(* CODESYS project BaseCodesys

Project tree, tasks and I/O mapping:
  Device : Berghof MC-PI SoftMotion Control , Berghof Automation GmbH, version 1.2.1.0
    application Application
      libraries: Standard, 3.5.18.0 (System); VisuDialogs, * (System)
      task EtherCAT_Task (cyclic, interval 1 ms, priority 0) calls PLC_PRG, POU
      task VISU_TASK (cyclic, interval 100 ms, priority 31) calls VisuElems.Visu_Prg
      program PLC_PRG [LD]
      trace Suivi (task EtherCAT_Task): PLC_PRG.MC_ReadActualPosition_0.Position
      Symbols
    EtherCAT_Master_SoftMotion : EtherCAT Master SoftMotion, 3S - Smart Software Solutions GmbH, version 4.4.0.0
        settings: MasterCycleTime = 1000; SlaveAutoRestart = True; NetworkName = 'eth0'; NetworkName = "eth0"; SrcAddress1 = 58463; SrcAddress2 = 30116746
      SC6_1 : SI6_SC6_DoubleAx_SoftMotion, STOEBER ANTRIEBSTECHNIK GmbH & Co. KG, version 4.5.0.0
          settings: ModularDevice = True; Number of Outputs = 0; Number of Inputs = 0; Number of Infos about Outputs = 0; Number of Infos about Inputs = 0; EnableExpertSettings = True; MDP_InputOffsets = [0,0,232]; MDP_OutputOffsets = [0,0,184]; StationAlias = 1002; Optional = False; DeviceIdenticationADO = 0; DeviceIdenticationMode = 0; Sync.Length = 46; Sync.Length = 58; FMMU.Length = 46; FMMU.Length = 58; Number of RxPDOs of the Slave = 2; Number of TxPDOs of the Slave = 2; DC sync0 cycletime = 1000; DC sync1 cycletime = 1000; EoEEnabled = True; EoEVirtualMACID = [16#02,16#01,16#05,16#10,16#03,16#E9]; EoEIPPortEnabled = False; EoEIPAddress = [16#00,16#00,16#00,16#00]; EoESubnetMask = [16#00,16#00,16#00,16#00]; EoEDefaultGateway = [16#00,16#00,16#00,16#00]; EoEDNSServer = [16#00,16#00,16#00,16#00]; EoEDNSName = 'SC6_1'; RxTxPdo.NumberofExcludes = 0; RxTxPdo.NumberofEntries = 8; RxTxPdo.Index = 16#1600; RxTxPdo.Fixed = False; RxTxPdo.Mandatory = False; RxTxPdo.Virtual = False; RxTxPdo.Sm = 2; RxTxPdo.Su = 0; RxTxPdo.Name = 'Axis A to Slave'; RxTxPdo.DependOnSlot = False; RxTxPdo.DependOnSlotGroup = False; RxTxPdo.OverwrittenByModule = True;
            A515 Controlword.Index = 16#6040; A515 Controlword.SubIndex = 0; A515 Controlword.Size = 16; A515 Controlword.Offset = 0; A515 Controlword.DependOnSlot = False; A515 Controlword.DependOnSlotGroup = False; A541 Modes of operation.Index = 16#6060; A541 Modes of operation.SubIndex = 0; A541 Modes of operation.Size = 8; A541 Modes of operation.Offset = 0; A541 Modes of operation.DependOnSlot = False; A541 Modes of operation.DependOnSlotGroup = False; A567 Target position.Index = 16#607A; A567 Target position.SubIndex = 0; A567 Target position.Size = 32; A567 Target position.Offset = 0; A567 Target position.DependOnSlot = False; A567 Target position.DependOnSlotGroup = False; A638 Target velocity.Index = 16#60FF; A638 Target velocity.SubIndex = 0; A638 Target velocity.Size = 32; A638 Target velocity.Offset = 0; A638 Target velocity.DependOnSlot = False; A638 Target velocity.DependOnSlotGroup = False; A592 Velocity offset.Index = 16#60B1; A592 Velocity offset.SubIndex = 0; A592 Velocity offset.Size = 32; A592 Velocity offset.Offset = 0; A592 Velocity offset.DependOnSlot = False; A592 Velocity offset.DependOnSlotGroup = False; A593 Torque offset.Index = 16#60B2; A593 Torque offset.SubIndex = 0; A593 Torque offset.Size = 16; A593 Torque offset.Offset = 0; A593 Torque offset.DependOnSlot = False; A593 Torque offset.DependOnSlotGroup = False; A558 Target torque.Index = 16#6071; A558 Target torque.SubIndex = 0; A558 Target torque.Size = 16; A558 Target torque.Offset = 0;
            A558 Target torque.DependOnSlot = False; A558 Target torque.DependOnSlotGroup = False; A637 Digital outputs.Index = 16#60FE; A637 Digital outputs.SubIndex = 1; A637 Digital outputs.Size = 32; A637 Digital outputs.Offset = 0; A637 Digital outputs.DependOnSlot = False; A637 Digital outputs.DependOnSlotGroup = False; RxTxPdo.NumberofExcludes = 0; RxTxPdo.NumberofEntries = 8; RxTxPdo.Index = 16#1601; RxTxPdo.Fixed = False; RxTxPdo.Mandatory = False; RxTxPdo.Virtual = False; RxTxPdo.Sm = 2; RxTxPdo.Su = 0; RxTxPdo.Name = 'Axis B to Slave'; RxTxPdo.DependOnSlot = False; RxTxPdo.DependOnSlotGroup = False; RxTxPdo.OverwrittenByModule = True; 2.A515 Controlword.Index = 16#6840; 2.A515 Controlword.SubIndex = 0; 2.A515 Controlword.Size = 16; 2.A515 Controlword.Offset = 0; 2.A515 Controlword.DependOnSlot = False; 2.A515 Controlword.DependOnSlotGroup = False; 2.A541 Modes of operation.Index = 16#6860; 2.A541 Modes of operation.SubIndex = 0; 2.A541 Modes of operation.Size = 8; 2.A541 Modes of operation.Offset = 0; 2.A541 Modes of operation.DependOnSlot = False; 2.A541 Modes of operation.DependOnSlotGroup = False; 2.A567 Target position.Index = 16#687A; 2.A567 Target position.SubIndex = 0; 2.A567 Target position.Size = 32; 2.A567 Target position.Offset = 0; 2.A567 Target position.DependOnSlot = False; 2.A567 Target position.DependOnSlotGroup = False; 2.A638 Target velocity.Index = 16#68FF; 2.A638 Target velocity.SubIndex = 0;
            2.A638 Target velocity.Size = 32; 2.A638 Target velocity.Offset = 0; 2.A638 Target velocity.DependOnSlot = False; 2.A638 Target velocity.DependOnSlotGroup = False; 2.A592 Velocity offset.Index = 16#68B1; 2.A592 Velocity offset.SubIndex = 0; 2.A592 Velocity offset.Size = 32; 2.A592 Velocity offset.Offset = 0; 2.A592 Velocity offset.DependOnSlot = False; 2.A592 Velocity offset.DependOnSlotGroup = False; 2.A593 Torque offset.Index = 16#68B2; 2.A593 Torque offset.SubIndex = 0; 2.A593 Torque offset.Size = 16; 2.A593 Torque offset.Offset = 0; 2.A593 Torque offset.DependOnSlot = False; 2.A593 Torque offset.DependOnSlotGroup = False; 2.A558 Target torque.Index = 16#6871; 2.A558 Target torque.SubIndex = 0; 2.A558 Target torque.Size = 16; 2.A558 Target torque.Offset = 0; 2.A558 Target torque.DependOnSlot = False; 2.A558 Target torque.DependOnSlotGroup = False; 2.A637 Digital outputs.Index = 16#68FE; 2.A637 Digital outputs.SubIndex = 1; 2.A637 Digital outputs.Size = 32; 2.A637 Digital outputs.Offset = 0; 2.A637 Digital outputs.DependOnSlot = False; 2.A637 Digital outputs.DependOnSlotGroup = False; RxTxPdo.NumberofExcludes = 0; RxTxPdo.NumberofEntries = 10; RxTxPdo.Index = 16#1A00; RxTxPdo.Fixed = False; RxTxPdo.Mandatory = False; RxTxPdo.Virtual = False; RxTxPdo.Sm = 3; RxTxPdo.Su = 0; RxTxPdo.Name = 'Axis A to Master'; RxTxPdo.DependOnSlot = False; RxTxPdo.DependOnSlotGroup = False; RxTxPdo.OverwrittenByModule = True;
            A516 Statusword.Index = 16#6041; A516 Statusword.SubIndex = 0; A516 Statusword.Size = 16; A516 Statusword.Offset = 0; A516 Statusword.DependOnSlot = False; A516 Statusword.DependOnSlotGroup = False; A542 Modes of operation display.Index = 16#6061; A542 Modes of operation display.SubIndex = 0; A542 Modes of operation display.Size = 8; A542 Modes of operation display.Offset = 0; A542 Modes of operation display.DependOnSlot = False; A542 Modes of operation display.DependOnSlotGroup = False; A545 Position actual value.Index = 16#6064; A545 Position actual value.SubIndex = 0; A545 Position actual value.Size = 32; A545 Position actual value.Offset = 0; A545 Position actual value.DependOnSlot = False; A545 Position actual value.DependOnSlotGroup = False; A553 Velocity actual value.Index = 16#606C; A553 Velocity actual value.SubIndex = 0; A553 Velocity actual value.Size = 32; A553 Velocity actual value.Offset = 0; A553 Velocity actual value.DependOnSlot = False; A553 Velocity actual value.DependOnSlotGroup = False; A564 Torque actual value.Index = 16#6077; A564 Torque actual value.SubIndex = 0; A564 Torque actual value.Size = 16; A564 Torque actual value.Offset = 0; A564 Torque actual value.DependOnSlot = False; A564 Torque actual value.DependOnSlotGroup = False; A632 Following error actual value.Index = 16#60F4; A632 Following error actual value.SubIndex = 0; A632 Following error actual value.Size = 32; A632 Following error actual value.Offset = 0; A632 Following error actual value.DependOnSlot = False; A632 Following error actual value.DependOnSlotGroup = False; A636 Digital inputs.Index = 16#60FD; A636 Digital inputs.SubIndex = 0; A636 Digital inputs.Size = 32; A636 Digital inputs.Offset = 0;
            A636 Digital inputs.DependOnSlot = False; A636 Digital inputs.DependOnSlotGroup = False; A620 Additional position actual value / 1st value.Index = 16#60E4; A620 Additional position actual value / 1st value.SubIndex = 1; A620 Additional position actual value / 1st value.Size = 32; A620 Additional position actual value / 1st value.Offset = 0; A620 Additional position actual value / 1st value.DependOnSlot = False; A620 Additional position actual value / 1st value.DependOnSlotGroup = False; E201 Statuswort 2.Index = 16#28C9; E201 Statuswort 2.SubIndex = 0; E201 Statuswort 2.Size = 16; E201 Statuswort 2.Offset = 0; E201 Statuswort 2.DependOnSlot = False; E201 Statuswort 2.DependOnSlotGroup = False; A67 User Statuswort.Index = 16#2043; A67 User Statuswort.SubIndex = 0; A67 User Statuswort.Size = 16; A67 User Statuswort.Offset = 0; A67 User Statuswort.DependOnSlot = False; A67 User Statuswort.DependOnSlotGroup = False; RxTxPdo.NumberofExcludes = 0; RxTxPdo.NumberofEntries = 10; RxTxPdo.Index = 16#1A01; RxTxPdo.Fixed = False; RxTxPdo.Mandatory = False; RxTxPdo.Virtual = False; RxTxPdo.Sm = 3; RxTxPdo.Su = 0; RxTxPdo.Name = 'Axis B to Master'; RxTxPdo.DependOnSlot = False; RxTxPdo.DependOnSlotGroup = False; RxTxPdo.OverwrittenByModule = True; 2.A516 Statusword.Index = 16#6841; 2.A516 Statusword.SubIndex = 0; 2.A516 Statusword.Size = 16; 2.A516 Statusword.Offset = 0; 2.A516 Statusword.DependOnSlot = False; 2.A516 Statusword.DependOnSlotGroup = False; 2.A542 Modes of operation display.Index = 16#6861; 2.A542 Modes of operation display.SubIndex = 0;
            2.A542 Modes of operation display.Size = 8; 2.A542 Modes of operation display.Offset = 0; 2.A542 Modes of operation display.DependOnSlot = False; 2.A542 Modes of operation display.DependOnSlotGroup = False; 2.A545 Position actual value.Index = 16#6864; 2.A545 Position actual value.SubIndex = 0; 2.A545 Position actual value.Size = 32; 2.A545 Position actual value.Offset = 0; 2.A545 Position actual value.DependOnSlot = False; 2.A545 Position actual value.DependOnSlotGroup = False; 2.A553 Velocity actual value.Index = 16#686C; 2.A553 Velocity actual value.SubIndex = 0; 2.A553 Velocity actual value.Size = 32; 2.A553 Velocity actual value.Offset = 0; 2.A553 Velocity actual value.DependOnSlot = False; 2.A553 Velocity actual value.DependOnSlotGroup = False; 2.A564 Torque actual value.Index = 16#6877; 2.A564 Torque actual value.SubIndex = 0; 2.A564 Torque actual value.Size = 16; 2.A564 Torque actual value.Offset = 0; 2.A564 Torque actual value.DependOnSlot = False; 2.A564 Torque actual value.DependOnSlotGroup = False; 2.A632 Following error actual value.Index = 16#68F4; 2.A632 Following error actual value.SubIndex = 0; 2.A632 Following error actual value.Size = 32; 2.A632 Following error actual value.Offset = 0; 2.A632 Following error actual value.DependOnSlot = False; 2.A632 Following error actual value.DependOnSlotGroup = False; 2.636 Digital inputs.Index = 16#68FD; 2.636 Digital inputs.SubIndex = 0; 2.636 Digital inputs.Size = 32; 2.636 Digital inputs.Offset = 0; 2.636 Digital inputs.DependOnSlot = False; 2.636 Digital inputs.DependOnSlotGroup = False; 2.A620 Additional position actual value / 1st value.Index = 16#68E4; 2.A620 Additional position actual value / 1st value.SubIndex = 1; 2.A620 Additional position actual value / 1st value.Size = 32; 2.A620 Additional position actual value / 1st value.Offset = 0; 2.A620 Additional position actual value / 1st value.DependOnSlot = False; 2.A620 Additional position actual value / 1st value.DependOnSlotGroup = False;
            2.E201 Statuswort 2.Index = 16#A8C9; 2.E201 Statuswort 2.SubIndex = 0; 2.E201 Statuswort 2.Size = 16; 2.E201 Statuswort 2.Offset = 0; 2.E201 Statuswort 2.DependOnSlot = False; 2.E201 Statuswort 2.DependOnSlotGroup = False; 2.A67 User Statuswort.Index = 16#A043; 2.A67 User Statuswort.SubIndex = 0; 2.A67 User Statuswort.Size = 16; 2.A67 User Statuswort.Offset = 0; 2.A67 User Statuswort.DependOnSlot = False; 2.A67 User Statuswort.DependOnSlotGroup = False; A515 Controlword.Name = 'A515 Controlword'; A515 Controlword.DataType = 'WORD'; A515 Controlword.Default = ''; A515 Controlword.Comment = ''; A541 Modes of operation.Name = 'A541 Modes of operation'; A541 Modes of operation.DataType = 'SINT'; A541 Modes of operation.Default = ''; A541 Modes of operation.Comment = ''; A567 Target position.Name = 'A567 Target position'; A567 Target position.DataType = 'DINT'; A567 Target position.Default = ''; A567 Target position.Comment = ''; A638 Target velocity.Name = 'A638 Target velocity'; A638 Target velocity.DataType = 'DINT'; A638 Target velocity.Default = ''; A638 Target velocity.Comment = ''; A592 Velocity offset.Name = 'A592 Velocity offset'; A592 Velocity offset.DataType = 'DINT'; A592 Velocity offset.Default = ''; A592 Velocity offset.Comment = ''; A593 Torque offset.Name = 'A593 Torque offset'; A593 Torque offset.DataType = 'INT'; A593 Torque offset.Default = ''; A593 Torque offset.Comment = ''; A558 Target torque.Name = 'A558 Target torque'; A558 Target torque.DataType = 'INT'; A558 Target torque.Default = ''; A558 Target torque.Comment = '';
            A637 Digital outputs.Name = 'A637 Digital outputs'; A637 Digital outputs.DataType = 'DWORD'; A637 Digital outputs.Default = ''; A637 Digital outputs.Comment = ''; 2.A515 Controlword.Name = '2.A515 Controlword'; 2.A515 Controlword.DataType = 'WORD'; 2.A515 Controlword.Default = ''; 2.A515 Controlword.Comment = ''; 2.A541 Modes of operation.Name = '2.A541 Modes of operation'; 2.A541 Modes of operation.DataType = 'SINT'; 2.A541 Modes of operation.Default = ''; 2.A541 Modes of operation.Comment = ''; 2.A567 Target position.Name = '2.A567 Target position'; 2.A567 Target position.DataType = 'DINT'; 2.A567 Target position.Default = ''; 2.A567 Target position.Comment = ''; 2.A638 Target velocity.Name = '2.A638 Target velocity'; 2.A638 Target velocity.DataType = 'DINT'; 2.A638 Target velocity.Default = ''; 2.A638 Target velocity.Comment = ''; 2.A592 Velocity offset.Name = '2.A592 Velocity offset'; 2.A592 Velocity offset.DataType = 'DINT'; 2.A592 Velocity offset.Default = ''; 2.A592 Velocity offset.Comment = ''; 2.A593 Torque offset.Name = '2.A593 Torque offset'; 2.A593 Torque offset.DataType = 'INT'; 2.A593 Torque offset.Default = ''; 2.A593 Torque offset.Comment = ''; 2.A558 Target torque.Name = '2.A558 Target torque'; 2.A558 Target torque.DataType = 'INT'; 2.A558 Target torque.Default = ''; 2.A558 Target torque.Comment = ''; 2.A637 Digital outputs.Name = '2.A637 Digital outputs'; 2.A637 Digital outputs.DataType = 'DWORD'; 2.A637 Digital outputs.Default = ''; 2.A637 Digital outputs.Comment = ''; A516 Statusword.Name = 'A516 Statusword'; A516 Statusword.DataType = 'WORD'; A516 Statusword.Default = ''; A516 Statusword.Comment = '';
            A542 Modes of operation display.Name = 'A542 Modes of operation display'; A542 Modes of operation display.DataType = 'SINT'; A542 Modes of operation display.Default = ''; A542 Modes of operation display.Comment = ''; A545 Position actual value.Name = 'A545 Position actual value'; A545 Position actual value.DataType = 'DINT'; A545 Position actual value.Default = ''; A545 Position actual value.Comment = ''; A553 Velocity actual value.Name = 'A553 Velocity actual value'; A553 Velocity actual value.DataType = 'DINT'; A553 Velocity actual value.Default = ''; A553 Velocity actual value.Comment = ''; A564 Torque actual value.Name = 'A564 Torque actual value'; A564 Torque actual value.DataType = 'INT'; A564 Torque actual value.Default = ''; A564 Torque actual value.Comment = ''; A632 Following error actual value.Name = 'A632 Following error actual value'; A632 Following error actual value.DataType = 'DINT'; A632 Following error actual value.Default = ''; A632 Following error actual value.Comment = ''; A636 Digital inputs.Name = 'A636 Digital inputs'; A636 Digital inputs.DataType = 'DWORD'; A636 Digital inputs.Default = ''; A636 Digital inputs.Comment = ''; A620 Additional position actual value / 1st value.Name = 'A620 Additional position actual value / 1st value'; A620 Additional position actual value / 1st value.DataType = 'DINT'; A620 Additional position actual value / 1st value.Default = ''; A620 Additional position actual value / 1st value.Comment = ''; E201 Statuswort 2.Name = 'E201 Statuswort 2'; E201 Statuswort 2.DataType = 'WORD'; E201 Statuswort 2.Default = ''; E201 Statuswort 2.Comment = ''; A67 User Statuswort.Name = 'A67 User Statuswort'; A67 User Statuswort.DataType = 'WORD'; A67 User Statuswort.Default = ''; A67 User Statuswort.Comment = ''; 2.A516 Statusword.Name = '2.A516 Statusword'; 2.A516 Statusword.DataType = 'WORD'; 2.A516 Statusword.Default = ''; 2.A516 Statusword.Comment = '';
            2.A542 Modes of operation display.Name = '2.A542 Modes of operation display'; 2.A542 Modes of operation display.DataType = 'SINT'; 2.A542 Modes of operation display.Default = ''; 2.A542 Modes of operation display.Comment = ''; 2.A545 Position actual value.Name = '2.A545 Position actual value'; 2.A545 Position actual value.DataType = 'DINT'; 2.A545 Position actual value.Default = ''; 2.A545 Position actual value.Comment = ''; 2.A553 Velocity actual value.Name = '2.A553 Velocity actual value'; 2.A553 Velocity actual value.DataType = 'DINT'; 2.A553 Velocity actual value.Default = ''; 2.A553 Velocity actual value.Comment = ''; 2.A564 Torque actual value.Name = '2.A564 Torque actual value'; 2.A564 Torque actual value.DataType = 'INT'; 2.A564 Torque actual value.Default = ''; 2.A564 Torque actual value.Comment = ''; 2.A632 Following error actual value.Name = '2.A632 Following error actual value'; 2.A632 Following error actual value.DataType = 'DINT'; 2.A632 Following error actual value.Default = ''; 2.A632 Following error actual value.Comment = ''; 2.636 Digital inputs.Name = '2.636 Digital inputs'; 2.636 Digital inputs.DataType = 'DWORD'; 2.636 Digital inputs.Default = ''; 2.636 Digital inputs.Comment = ''; 2.A620 Additional position actual value / 1st value.Name = '2.A620 Additional position actual value / 1st value'; 2.A620 Additional position actual value / 1st value.DataType = 'DINT'; 2.A620 Additional position actual value / 1st value.Default = ''; 2.A620 Additional position actual value / 1st value.Comment = ''; 2.E201 Statuswort 2.Name = '2.E201 Statuswort 2'; 2.E201 Statuswort 2.DataType = 'WORD'; 2.E201 Statuswort 2.Default = ''; 2.E201 Statuswort 2.Comment = ''; 2.A67 User Statuswort.Name = '2.A67 User Statuswort'; 2.A67 User Statuswort.DataType = 'WORD'; 2.A67 User Statuswort.Default = ''; 2.A67 User Statuswort.Comment = ''
        CiA_ControllerBased : xA CBM_SoftMotion, STOEBER ANTRIEBSTECHNIK GmbH & Co. KG, version 4.4.0.0
            settings: Number of Outputs = 8; Number of Inputs = 10; Number of Infos about Outputs = 8; Number of Infos about Inputs = 10; RxTxPdo.Mandatory = False; RxTxPdo.Virtual = False; RxTxPdo.DependOnSlot = False; RxTxPdo.DependOnSlotGroup = False; A515 Controlword.Offset = 0; A515 Controlword.DependOnSlot = False; A515 Controlword.DependOnSlotGroup = False; A541 Modes of operation.Offset = 0; A541 Modes of operation.DependOnSlot = False; A541 Modes of operation.DependOnSlotGroup = False; A567 Target position.Offset = 0; A567 Target position.DependOnSlot = False; A567 Target position.DependOnSlotGroup = False; A638 Target velocity.Offset = 0; A638 Target velocity.DependOnSlot = False; A638 Target velocity.DependOnSlotGroup = False; A592 Velocity offset.Offset = 0; A592 Velocity offset.DependOnSlot = False; A592 Velocity offset.DependOnSlotGroup = False; A593 Torque offset.Offset = 0; A593 Torque offset.DependOnSlot = False; A593 Torque offset.DependOnSlotGroup = False; A558 Target torque.Offset = 0; A558 Target torque.DependOnSlot = False; A558 Target torque.DependOnSlotGroup = False; A637 Digital outputs.Offset = 0; A637 Digital outputs.DependOnSlot = False; A637 Digital outputs.DependOnSlotGroup = False; RxTxPdo.Mandatory = False; RxTxPdo.Virtual = False; RxTxPdo.DependOnSlot = False; RxTxPdo.DependOnSlotGroup = False; A516 Statusword.Offset = 0; A516 Statusword.DependOnSlot = False; A516 Statusword.DependOnSlotGroup = False; A542 Modes of operation display.Offset = 0;
              A542 Modes of operation display.DependOnSlot = False; A542 Modes of operation display.DependOnSlotGroup = False; A545 Position actual value.Offset = 0; A545 Position actual value.DependOnSlot = False; A545 Position actual value.DependOnSlotGroup = False; A553 Velocity actual value.Offset = 0; A553 Velocity actual value.DependOnSlot = False; A553 Velocity actual value.DependOnSlotGroup = False; A564 Torque actual value.Offset = 0; A564 Torque actual value.DependOnSlot = False; A564 Torque actual value.DependOnSlotGroup = False; A632 Following error actual value.Offset = 0; A632 Following error actual value.DependOnSlot = False; A632 Following error actual value.DependOnSlotGroup = False; A636 Digital inputs.Offset = 0; A636 Digital inputs.DependOnSlot = False; A636 Digital inputs.DependOnSlotGroup = False; A620 Additional position actual value / 1st value.Offset = 0; A620 Additional position actual value / 1st value.DependOnSlot = False; A620 Additional position actual value / 1st value.DependOnSlotGroup = False; E201 Statuswort 2.Offset = 0; E201 Statuswort 2.DependOnSlot = False; E201 Statuswort 2.DependOnSlotGroup = False; A67 User Statuswort.Offset = 0; A67 User Statuswort.DependOnSlot = False; A67 User Statuswort.DependOnSlotGroup = False; A515 Controlword.Default = ''; A541 Modes of operation.Default = ''; A567 Target position.Default = ''; A638 Target velocity.Default = ''; A592 Velocity offset.Default = ''; A593 Torque offset.Default = ''; A558 Target torque.Default = ''; A637 Digital outputs.Default = ''; A516 Statusword.Default = ''; A542 Modes of operation display.Default = ''; A545 Position actual value.Default = ''; A553 Velocity actual value.Default = ''; A564 Torque actual value.Default = ''; A632 Following error actual value.Default = '';
              A636 Digital inputs.Default = ''; A620 Additional position actual value / 1st value.Default = ''; E201 Statuswort 2.Default = ''; A67 User Statuswort.Default = ''
            unmapped channels: A515 Controlword, A541 Modes of operation, A567 Target position, A638 Target velocity, A592 Velocity offset, A593 Torque offset, A558 Target torque, A637 Digital outputs, A516 Statusword, A542 Modes of operation display, A545 Position actual value, A553 Velocity actual value, A564 Torque actual value, A632 Following error actual value, A636 Digital inputs, A620 Additional position actual value / 1st value, E201 Statuswort 2, A67 User Statuswort
        CiA_ControllerBased_1 : xB CBM_SoftMotion, STOEBER ANTRIEBSTECHNIK GmbH & Co. KG, version 4.4.0.0
            settings: Number of Outputs = 8; Number of Inputs = 10; Number of Infos about Outputs = 8; Number of Infos about Inputs = 10; RxTxPdo.Mandatory = False; RxTxPdo.Virtual = False; RxTxPdo.DependOnSlot = False; RxTxPdo.DependOnSlotGroup = False; 2.A515 Controlword.Offset = 0; 2.A515 Controlword.DependOnSlot = False; 2.A515 Controlword.DependOnSlotGroup = False; 2.A541 Modes of operation.Offset = 0; 2.A541 Modes of operation.DependOnSlot = False; 2.A541 Modes of operation.DependOnSlotGroup = False; 2.A567 Target position.Offset = 0; 2.A567 Target position.DependOnSlot = False; 2.A567 Target position.DependOnSlotGroup = False; 2.A638 Target velocity.Offset = 0; 2.A638 Target velocity.DependOnSlot = False; 2.A638 Target velocity.DependOnSlotGroup = False; 2.A592 Velocity offset.Offset = 0; 2.A592 Velocity offset.DependOnSlot = False; 2.A592 Velocity offset.DependOnSlotGroup = False; 2.A593 Torque offset.Offset = 0; 2.A593 Torque offset.DependOnSlot = False; 2.A593 Torque offset.DependOnSlotGroup = False; 2.A558 Target torque.Offset = 0; 2.A558 Target torque.DependOnSlot = False; 2.A558 Target torque.DependOnSlotGroup = False; 2.A637 Digital outputs.Offset = 0; 2.A637 Digital outputs.DependOnSlot = False; 2.A637 Digital outputs.DependOnSlotGroup = False; RxTxPdo.Mandatory = False; RxTxPdo.Virtual = False; RxTxPdo.DependOnSlot = False; RxTxPdo.DependOnSlotGroup = False; 2.A516 Statusword.Offset = 0; 2.A516 Statusword.DependOnSlot = False; 2.A516 Statusword.DependOnSlotGroup = False; 2.A542 Modes of operation display.Offset = 0;
              2.A542 Modes of operation display.DependOnSlot = False; 2.A542 Modes of operation display.DependOnSlotGroup = False; 2.A545 Position actual value.Offset = 0; 2.A545 Position actual value.DependOnSlot = False; 2.A545 Position actual value.DependOnSlotGroup = False; 2.A553 Velocity actual value.Offset = 0; 2.A553 Velocity actual value.DependOnSlot = False; 2.A553 Velocity actual value.DependOnSlotGroup = False; 2.A564 Torque actual value.Offset = 0; 2.A564 Torque actual value.DependOnSlot = False; 2.A564 Torque actual value.DependOnSlotGroup = False; 2.A632 Following error actual value.Offset = 0; 2.A632 Following error actual value.DependOnSlot = False; 2.A632 Following error actual value.DependOnSlotGroup = False; 2.636 Digital inputs.Index = 16#68FD; 2.636 Digital inputs.SubIndex = 0; 2.636 Digital inputs.Size = 32; 2.636 Digital inputs.Offset = 0; 2.636 Digital inputs.DependOnSlot = False; 2.636 Digital inputs.DependOnSlotGroup = False; 2.A620 Additional position actual value / 1st value.Offset = 0; 2.A620 Additional position actual value / 1st value.DependOnSlot = False; 2.A620 Additional position actual value / 1st value.DependOnSlotGroup = False; 2.E201 Statuswort 2.Offset = 0; 2.E201 Statuswort 2.DependOnSlot = False; 2.E201 Statuswort 2.DependOnSlotGroup = False; 2.A67 User Statuswort.Offset = 0; 2.A67 User Statuswort.DependOnSlot = False; 2.A67 User Statuswort.DependOnSlotGroup = False; 2.A515 Controlword.Default = ''; 2.A541 Modes of operation.Default = ''; 2.A567 Target position.Default = ''; 2.A638 Target velocity.Default = ''; 2.A592 Velocity offset.Default = ''; 2.A593 Torque offset.Default = ''; 2.A558 Target torque.Default = ''; 2.A637 Digital outputs.Default = ''; 2.A516 Statusword.Default = ''; 2.A542 Modes of operation display.Default = ''; 2.A545 Position actual value.Default = '';
              2.A553 Velocity actual value.Default = ''; 2.A564 Torque actual value.Default = ''; 2.A632 Following error actual value.Default = ''; 2.636 Digital inputs.Name = '2.636 Digital inputs'; 2.636 Digital inputs.DataType = 'DWORD'; 2.636 Digital inputs.Default = ''; 2.636 Digital inputs.Comment = ''; 2.A620 Additional position actual value / 1st value.Default = ''; 2.E201 Statuswort 2.Default = ''; 2.A67 User Statuswort.Default = ''
            unmapped channels: 2.A515 Controlword, 2.A541 Modes of operation, 2.A567 Target position, 2.A638 Target velocity, 2.A592 Velocity offset, 2.A593 Torque offset, 2.A558 Target torque, 2.A637 Digital outputs, 2.A516 Statusword, 2.A542 Modes of operation display, 2.A545 Position actual value, 2.A553 Velocity actual value, 2.A564 Torque actual value, 2.A632 Following error actual value, 2.636 Digital inputs, 2.A620 Additional position actual value / 1st value, 2.E201 Statuswort 2, 2.A67 User Statuswort
        Piston : SM_Drive_ETC_STOEBER_SI6_SC6, 3S - Smart Software Solutions GmbH, order no. 0, version 4.5.0.0
            settings: wDriveID = 0; dwRatioTechUnitsDenom = 131072; iRatioTechUnitsNum = 45; iMovementType = 0; fPositionPeriod = 360; fSWMaxVelocity = 36000; fSWMaxAcceleration = 30000; fSWMaxDeceleration = 30000; fSWMaxJerk = 30000; Commisioning.smci.Distance = 1048576; Commisioning.smci.Velocity = 2000; Commisioning.smci.Acceleration = 10000; Commisioning.smci.Deceleration = 10000; ScalingIncs = 1048576; ScalingUnits = 360; AdrOffset_8010 = 0; BitOffset_8010 = 0; BitLength_8010 = 16; Address_8010 = '%QW0'; Type_8010 = 'WORD'; AddressPointer_8010 = ADR(%QW0); AdrOffset_8020 = 4; BitOffset_8020 = 0; BitLength_8020 = 32; Address_8020 = '%QD1'; Type_8020 = 'DINT'; AddressPointer_8020 = ADR(%QD1); AdrOffset_8030 = 8; BitOffset_8030 = 0; BitLength_8030 = 32; Address_8030 = '%QD2'; Type_8030 = 'DINT'; AddressPointer_8030 = ADR(%QD2); AdrOffset_8040 = 18; BitOffset_8040 = 0; BitLength_8040 = 16; Address_8040 = '%QW9'; Type_8040 = 'INT'; AddressPointer_8040 = ADR(%QW9); AdrOffset_8050 = 2;
              BitOffset_8050 = 0; BitLength_8050 = 8; Address_8050 = '%QB2'; Type_8050 = 'SINT'; AddressPointer_8050 = ADR(%QB2); AdrOffset_8060 = 4294967295; BitOffset_8060 = 0; BitLength_8060 = 0; Address_8060 = ''; Type_8060 = ''; AddressPointer_8060 = 0; AdrOffset_8070 = 12; BitOffset_8070 = 0; BitLength_8070 = 32; Address_8070 = '%QD3'; Type_8070 = 'DINT'; AddressPointer_8070 = ADR(%QD3); AdrOffset_8080 = 16; BitOffset_8080 = 0; BitLength_8080 = 16; Address_8080 = '%QW8'; Type_8080 = 'INT'; AddressPointer_8080 = ADR(%QW8); AdrOffset_8090 = 20; BitOffset_8090 = 0; BitLength_8090 = 32; Address_8090 = '%QD5'; Type_8090 = 'DWORD'; AddressPointer_8090 = ADR(%QD5); AdrOffset_8510 = 0; BitOffset_8510 = 0; BitLength_8510 = 16; Address_8510 = '%IW0'; Type_8510 = 'WORD'; AddressPointer_8510 = ADR(%IW0); AdrOffset_8520 = 4; BitOffset_8520 = 0; BitLength_8520 = 32; Address_8520 = '%ID1'; Type_8520 = 'DINT';
              AddressPointer_8520 = ADR(%ID1); AdrOffset_8530 = 8; BitOffset_8530 = 0; BitLength_8530 = 32; Address_8530 = '%ID2'; Type_8530 = 'DINT'; AddressPointer_8530 = ADR(%ID2); AdrOffset_8540 = 12; BitOffset_8540 = 0; BitLength_8540 = 16; Address_8540 = '%IW6'; Type_8540 = 'INT'; AddressPointer_8540 = ADR(%IW6); AdrOffset_8550 = 2; BitOffset_8550 = 0; BitLength_8550 = 8; Address_8550 = '%IB2'; Type_8550 = 'SINT'; AddressPointer_8550 = ADR(%IB2); AdrOffset_8560 = 20; BitOffset_8560 = 0; BitLength_8560 = 32; Address_8560 = '%ID5'; Type_8560 = 'DWORD'; AddressPointer_8560 = ADR(%ID5); AdrOffset_8570 = 4294967295; BitOffset_8570 = 0; BitLength_8570 = 0; Address_8570 = ''; Type_8570 = ''; AddressPointer_8570 = 0; AdrOffset_8580 = 4294967295; BitOffset_8580 = 0; BitLength_8580 = 0; Address_8580 = ''; Type_8580 = ''; AddressPointer_8580 = 0; AdrOffset_8590 = 4294967295; BitOffset_8590 = 0; BitLength_8590 = 0;
              Address_8590 = ''; Type_8590 = ''; AddressPointer_8590 = 0; AdrOffset_8600 = 4294967295; BitOffset_8600 = 0; BitLength_8600 = 0; Address_8600 = ''; Type_8600 = ''; AddressPointer_8600 = 0; AdrOffset_8600 = 4294967295; BitOffset_8600 = 0; BitLength_8600 = 0; Address_8610 = ''; Type_8610 = ''; AddressPointer_8610 = 0; AdrOffset_8600 = 28; BitOffset_8600 = 0; BitLength_8600 = 16; Address_8620 = '%IW14'; Type_8620 = 'WORD'; AddressPointer_8620 = ADR(%IW14); AdrOffset_8630 = 16; BitOffset_8630 = 0; BitLength_8630 = 32; Address_8630 = '%ID4'; Type_8630 = 'DINT'; AddressPointer_8630 = ADR(%ID4)
        Virtuel : SM_Drive_ETC_STOEBER_SI6_SC6, 3S - Smart Software Solutions GmbH, order no. 0, version 4.5.0.0
            settings: bVirtual = TRUE; dwRatioTechUnitsDenom = 512; iRatioTechUnitsNum = 45; iMovementType = 0; fSWMaxVelocity = 3000; ScalingIncs = 4096; ScalingUnits = 360; AdrOffset_8010 = 24; BitOffset_8010 = 0; BitLength_8010 = 16; Address_8010 = '%QW12'; Type_8010 = 'WORD'; AddressPointer_8010 = ADR(%QW12); AdrOffset_8020 = 28; BitOffset_8020 = 0; BitLength_8020 = 32; Address_8020 = '%QD7'; Type_8020 = 'DINT'; AddressPointer_8020 = ADR(%QD7); AdrOffset_8030 = 32; BitOffset_8030 = 0; BitLength_8030 = 32; Address_8030 = '%QD8'; Type_8030 = 'DINT'; AddressPointer_8030 = ADR(%QD8); AdrOffset_8040 = 42; BitOffset_8040 = 0; BitLength_8040 = 16; Address_8040 = '%QW21'; Type_8040 = 'INT'; AddressPointer_8040 = ADR(%QW21); AdrOffset_8050 = 26; BitOffset_8050 = 0; BitLength_8050 = 8; Address_8050 = '%QB26'; Type_8050 = 'SINT'; AddressPointer_8050 = ADR(%QB26); AdrOffset_8060 = 4294967295; BitOffset_8060 = 0; BitLength_8060 = 0;
              Address_8060 = ''; Type_8060 = ''; AddressPointer_8060 = 0; AdrOffset_8070 = 36; BitOffset_8070 = 0; BitLength_8070 = 32; Address_8070 = '%QD9'; Type_8070 = 'DINT'; AddressPointer_8070 = ADR(%QD9); AdrOffset_8080 = 40; BitOffset_8080 = 0; BitLength_8080 = 16; Address_8080 = '%QW20'; Type_8080 = 'INT'; AddressPointer_8080 = ADR(%QW20); AdrOffset_8090 = 44; BitOffset_8090 = 0; BitLength_8090 = 32; Address_8090 = '%QD11'; Type_8090 = 'DWORD'; AddressPointer_8090 = ADR(%QD11); AdrOffset_8510 = 32; BitOffset_8510 = 0; BitLength_8510 = 16; Address_8510 = '%IW16'; Type_8510 = 'WORD'; AddressPointer_8510 = ADR(%IW16); AdrOffset_8520 = 36; BitOffset_8520 = 0; BitLength_8520 = 32; Address_8520 = '%ID9'; Type_8520 = 'DINT'; AddressPointer_8520 = ADR(%ID9); AdrOffset_8530 = 40; BitOffset_8530 = 0; BitLength_8530 = 32; Address_8530 = '%ID10'; Type_8530 = 'DINT'; AddressPointer_8530 = ADR(%ID10); AdrOffset_8540 = 44;
              BitOffset_8540 = 0; BitLength_8540 = 16; Address_8540 = '%IW22'; Type_8540 = 'INT'; AddressPointer_8540 = ADR(%IW22); AdrOffset_8550 = 34; BitOffset_8550 = 0; BitLength_8550 = 8; Address_8550 = '%IB34'; Type_8550 = 'SINT'; AddressPointer_8550 = ADR(%IB34); AdrOffset_8560 = 52; BitOffset_8560 = 0; BitLength_8560 = 32; Address_8560 = '%ID13'; Type_8560 = 'DWORD'; AddressPointer_8560 = ADR(%ID13); AdrOffset_8570 = 4294967295; BitOffset_8570 = 0; BitLength_8570 = 0; Address_8570 = ''; Type_8570 = ''; AddressPointer_8570 = 0; AdrOffset_8580 = 4294967295; BitOffset_8580 = 0; BitLength_8580 = 0; Address_8580 = ''; Type_8580 = ''; AddressPointer_8580 = 0; AdrOffset_8590 = 4294967295; BitOffset_8590 = 0; BitLength_8590 = 0; Address_8590 = ''; Type_8590 = ''; AddressPointer_8590 = 0; AdrOffset_8600 = 4294967295; BitOffset_8600 = 0; BitLength_8600 = 0; Address_8600 = ''; Type_8600 = '';
              AddressPointer_8600 = 0; AdrOffset_8600 = 4294967295; BitOffset_8600 = 0; BitLength_8600 = 0; Address_8610 = ''; Type_8610 = ''; AddressPointer_8610 = 0; AdrOffset_8600 = 60; BitOffset_8600 = 0; BitLength_8600 = 16; Address_8620 = '%IW30'; Type_8620 = 'WORD'; AddressPointer_8620 = ADR(%IW30); AdrOffset_8630 = 48; BitOffset_8630 = 0; BitLength_8630 = 32; Address_8630 = '%ID12'; Type_8630 = 'DINT'; AddressPointer_8630 = ADR(%ID12)
    Ethernet : Ethernet, 3S - Smart Software Solutions GmbH, version 4.1.0.0
        settings: IPAddress = [169,254,255,33]; SubnetMask = [255,255,255,0]; GatewayAddress = [0,0,0,0]; MACAddress = [16#00,16#E0,16#BA,16#A1,16#FF,16#F6]; NetworkInterfaceName = 'eth2'; NetworkInterfaceName = "eth2"; SaveCommunicationSettings = FALSE
      ModbusTCP_Slave_Device : ModbusTCP Slave Device, 3S - Smart Software Solutions GmbH, version 4.2.0.0
          settings: UpdateableHolding = TRUE; Coils Size = 16; Discrete Inputs Size = 16
          output Application.Gestion_axes.Gr_Piston.Mode_Asservi : BOOL  // Registres de retenue.Registres de retenue.Bit0
          output Application.Gestion_axes.Gr_Piston.Mvt_Avant : BOOL  // Registres de retenue.Registres de retenue.Bit1
          output Application.Gestion_axes.Gr_Piston.Mvt_Arriere : BOOL  // Registres de retenue.Registres de retenue.Bit2
          output Application.Gestion_axes.Gr_Piston.Mvt_Prise_Origine : BOOL  // Registres de retenue.Registres de retenue.Bit3
          output Application.Gestion_axes.Gr_Piston.Mvt_Aller_Position : BOOL  // Registres de retenue.Registres de retenue.Bit4
          output Application.GVL.clrfault : BOOL  // Registres de retenue.Registres de retenue.Bit5
          output Application.gestion_axes.Gr_Piston.Mvt_stop : BOOL  // Registres de retenue.Registres de retenue.Bit6
          output Application.gestion_axes.Gr_Piston.Mvt_Synchro : BOOL  // Registres de retenue.Registres de retenue.Bit7
          output Application.Gestion_axes.Gr_virtuel.Mode_Asservi : BOOL  // Registres de retenue.Registres de retenue.Bit8
          output Application.Gestion_axes.Gr_virtuel.Mvt_Avant : BOOL  // Registres de retenue.Registres de retenue.Bit9
          output Application.Gestion_axes.Gr_virtuel.Mvt_Arriere : BOOL  // Registres de retenue.Registres de retenue.Bit10
          output Application.Gestion_axes.Gr_virtuel.Mvt_Prise_Origine : BOOL  // Registres de retenue.Registres de retenue.Bit11
          output Application.Gestion_axes.Gr_virtuel.Mvt_Aller_Position : BOOL  // Registres de retenue.Registres de retenue.Bit12
          output Application.gestion_axes.Gr_virtuel.Mvt_stop : BOOL  // Registres de retenue.Registres de retenue.Bit13
          unmapped channels: Registres de retenue, Registres d’entrée
    SoftMotion General Axis Pool
      SMC_FreeEncoder : SMC_FreeEncoder, 3S - Smart Software Solutions GmbH, order no. 1805, version 3.5.5.0
          settings: wDriveID = 3; dwRatioTechUnitsDenom = 131072
      Virtuel_1 : SM_Drive_PosControl, 3S - Smart Software Solutions GmbH, order no. 1805, version 4.12.0.0
          settings: wDriveID = 2; bVirtual = TRUE; dwRatioTechUnitsDenom = 512; iRatioTechUnitsNum = 45; iMovementType = 0; fSWMaxVelocity = 8000; fSWMaxAcceleration = 100000; fSWMaxDeceleration = 10000; Commisioning.smci.Distance = 360; Commisioning.smci.Velocity = 1000; Commisioning.smci.Acceleration = 10000; Commisioning.smci.Deceleration = 10000; ScalingIncs = 4096; ScalingUnits = 360; IsLinearMotor = FALSE; MaximumOutputVelocityTU = 3600; MinimumOutputVelocityTU = -3600
  libraries: VisuSymbols, 4.1.0.0 (System); VisuDialogs, * (System)
  Accessoires/
    function block type_axe [ST]
  program AssignationAxesEtherCAT [ST]
  CNC
  program ConfigurationGenerale [ST]
  EtherCAT/
    function block EsclavesReady [ST]
    function block NombreEsclavesEtherCAT [ST]
    function block SlaveType [ST]
  Gestion axes/
    program Gestion_axes [LD]
    function block Gr_Axe [SFC]: Attente_active, Controlling_active, Homing_active, Jog_active, mapping_active, Move_Stop_position_active, Polling_active, SetChannelParameters_active, Stop_active
  text list GlobalTextList
  global variables GVL
  global variables GVL_EtherCAT
  data type info_axe
  global variables MC_Pi
  data type Parametres_axe
  Paramètres CNC
  program POU [LD]
  data type Specifiques_axe
  data type Status_axe
  Tests/
    program ChoixOpMode [ST]
  program TestsFonctions [ST]
  text list TextList
  data type Utilitaire_axe
  Utilitaires/
    function block Position_atteinte [LD]
  global variables var_infor
  global variables Var_PMC
  visualisation Visualization
  visualisation VisualizationAxe1
  visualisation VisualizationCamIn
  visualisation VisualizationVirtuel
*)

// info_axe
TYPE info_axe :
	
STRUCT

	
	(* ============   gestion erreur ===============*)
	iErrorNumber:INT;   (*    *)
	berror:BOOL;

	(* ============= type axe ===================*)
	bVirtuel: BOOL;
	bCodeur: BOOL;
	bDrive_PSSU_et_codeur_CAN: BOOL;
	bDrive_PSSU_et_codeur_PMCprimoC: BOOL;
	bDrive_CAN_Ethercat: BOOL;
	smoteur_utilise:STRING;
	
	
	(*=== *)
	diMotor_Speed_V:DINT;
	diMotor_MI2T:DINT;
	diDrive_DI2T:DINT;
	diDrive_I:DINT;
	difollowing_error_PE:DINT;
	diRotor_angle_PRD:DINT;
	diAmbient_temperature_TEMPE:DINT;  (* temperature dissipateur thermique en °C *)
	diHeatSink_temperature_TEMPH:DINT;  (* temperature ambiante  en °C *)
	diMotor_temperature_TEMPM:DINT;  (* temperature moteur    en Ohms *)
	diTension_VBUS:DINT;
	diTension_Min_VBUSMIN:DINT;
	dipower_supply_VBUSBAL:DINT;
	vbusecat:real;
		
END_STRUCT


END_TYPE

// Parametres_axe
TYPE Parametres_axe :
	
STRUCT
	sNom: STRING := 'avance_papier'; (* Nom de l'axe  dans la machine (Uniquement pour info Utilisateur) *)
	sMoteur: STRING := 'CODEUR'; (* Choix du moteur ou  'VIRTUEL' ou  'CODEUR'  (Voir dans Bibliothéque PILZ ; Bibliothéque Moteur ) *)
	udiResolution:UDINT:=8192;  (* résolution pour 1 tour codeur *)
	sTypeDeVariateur : STRING := 'ProtegoD';
	sBusDeComm : String := 'CAN'; (* CAN | ETHERCAT *)
	sChoixAxe: STRING := 'A'; (* Pour les variateurs double axes *)
	dwAdresseEtherCAT : DWORD := 1001 ; 
		
	(*udinumero: USINT := 1; (* Numero de l'axe ( sert de Chronologie de mise à jour des paramétres à la mise sous tension  ) *) *)
	structAxe:axis_ref_sm3;
	structMaitre:axis_ref_sm3;
	structMaitreDifferentiel:axis_ref_sm3;
	sNomMaitre:STRING;
	sNomMaitreDifferentiel:String;
	bCyclique:BOOL:=TRUE;
	diCycle: UDINT := 2110; (* pts     0=mouvement  Borné ( pas de Modulo)         (Distance en pts pour un cycle machine) {SB} *)

	rEchelle: REAL := 25.80; (*  4096 / 50/pi  Pts/mm ( 4096 pts / tour moteur quelque soit le retour moteur ou nbre pts codeur x 16) *)
	diContrainte_Mvt: DINT := 0; (* mm    0= Interdiction de mouvement en marche arriére ( ou Course Maxi si diCycle=0 ) *)
	diContrainte_Mvt_neg: DINT := 0;
	bSens: BOOL := 1; (* Choix du sens de rotation du moteur pour aller en avant (Ne jamais inversr les phases moteurs) {CW} *)
	bDirection_unique:BOOL:=FALSE; 
	rTolerance_poursuite_Maxi: REAL := 10; (* mm           ( Seuil d' erreur (# entre demande & réel ) imposant un arrêt asservissement {SE} *)
	
	(* ===== mouvement =====*)
	
	rvitesse:REAL;  (* en unités /sec *)
	rAcceleration: REAL := 21100; (* mm/sec²  (si = 2 x Vitesse => atteinte vitesse en 0.5 sec) {SA DC AA XA RC} *)
	rdecceleration: REAL :=21100; (* mm/sec²  (si = 2 x Vitesse => atteinte vitesse en 0.5 sec) {SA DC AA XA RC} *)
	rdecceleration_urgence: REAL :=21100; (* mm/sec²  (si = 2 x Vitesse => atteinte vitesse en 0.5 sec) {SA DC AA XA RC} *)
	rPosArret: REAL; (* mm                 (Choix de la position d'arrêt positionné) {ST position ou MA position} *)
	
	(* ============   registration ===============*)
	rCorrection_Registration: REAL := 5; (* mm    0=Pas de filtre fenêtre            (Fenêtre dans laquelle sera pris en compte l'origine) {SR} *)
	rFiltre_Registration: REAL := 5; (* mm    0=Pas de filtre fenêtre            (Fenêtre dans laquelle sera pris en compte l'origine) {FR} *)
	usiControle_Registration: USINT := 2; (* Nbre   0= Pas de contrôle   (Nombre de fois autorisée sans voir le capteur d'origine (en standard 2) {RT} *)
	rPosCapteur: REAL := 10; (* mm                (Position du compteur lors du passage à 1 du capteur d'origine ) {RF} *)
	
	(*============= embrayage  synchronisation ===*)
	rFenetre_Embrayage: REAL := 5; (* mm    0=OFF (Zone dans laquelle les axes esclaves seront réalignés) {CI} *)
	rDistance_Embrayage: REAL := 0; (* %Cycle Maître  si #0 =>embrayage à la volée (CL) si =0 => Alignement des axes *)
	rPhase_maitre: REAL := 0; (* Ratio de Cycle maître    (Valeur entre -1 & +1)          (Calage entre cet axe et son maître) {MB} *)
	stype_embrayage:STRING:='VOLEE';   (*   'VOLEE', 'ALIGNEMENT_COURT','ALIGNEMENT_AVANT','ALIGNEMENT_ARRIERE','VITESSE'   *)
	sLoi_MVT: STRING := 'papier'; (* Nom came ex: 'CAME1'    Synchro linéaire en position  'LINEAR'  Synchro linéaire en  vitesse  'VITESSE' *)
	
	
	
	Gain_vitesse: REAL := 16; (* Gain Vitesse  >>> Valeur à régler sur place : mettre 3 ,puis augmenter jusqu'au bruit ,,enfin réduire de 10% *)
	Frein: BOOL := 0; (* 0= Pas de frein 1= Avec Frein {"MBRAKE"} *)
	Tension_secteur: REAL := 1; (* Choix de tension Secteur ==> si DD5 ou protegoD:  1=220v 2=400v  3=480v         ==> si DD4:          0=220v 1=400v  2=480v             {"VBUSBAL"} *)
	Mode_Asservissement: USINT := 24; (* Si Tendo DD 24=Relatif , 26=absolu, si  PrimoDrive 0=Relatif  7=Absolu{FS} *)
	Mode_Asservissement_secondaire:USINT:=0; (*Lorsque l'on va potentiellement faire varier le FS pendant le process, on indique ici le second FS qui sera utilisé *)
	

	

END_STRUCT


END_TYPE

// Specifiques_axe
TYPE Specifiques_axe :
	
STRUCT

	
	(* ============   codeur ===============*)
	Boucle_codeur_externe:BOOL; (* Si on souhaite utiliser un codeur branché sur le contrôleur pour fermer la boucle de position et non pas le retour de mesure du moteur *)
	Changement_Feedback_possible:BOOL; (* True si on souhaite pouvoir changer de retour de mesure. Tantôt avec le retour du moteur, tantôt par un codeur externe *)
	Channel_codeur_externe:USINT; (* Axe sur lequel on a défini le codeur externe CD 27 *)
	Multiplication_points_codeur:USINT:=2;   (*   la resolution est multipliée par 2^MS     si MS 4  ==> multiplication par 16 *)
	Filtre_codeur:UINT:=4;  (*  filtrage du signal codeur en faisant une moyenne sur le temps PT en msec *)
	
	(* ======== Mode Entrée ou Sortie ======= *)
	INOut1_X3A_6:BOOL;   (*  si 1  ==> borne X3A_6   gérée en entrée (O1MODE23)                 si 0  ==> borne X3A_6   gérée en sortie (O1MODE0)  *)
	INOut2_X3A_6:BOOL;   (*  si 1  ==> borne X3A_6   gérée en entrée (O1MODE23)                 si 0  ==> borne X3A_6   gérée en sortie (O1MODE0)  *)
	
   (* ==== Gain intégral boucle de vitesse ==== *)
   (* valeur en msec de base à 10 *)
   (* Smaller motors permit shorter integration times. Larger motors or high moments of inertia in the load usually require integration times of 20ms or more. *)
   (* With GVTN=0ms, the I-component is switched off. If the GVTN value is too low, the drive runs roughly or strongly overshoots with high inertia loads. *)
   (*  If the GVTN value is too high, the drive is too soft. *)
   Gain_integral_vitesse:REAL:=10;
   
    (* ==== Gain boucle de position ==== *)
	Gain_position:REAL:=0.1;
	
	 (* ==== mapping ==== *)
	 Phase_esclave:REAL;     (* MF *)
	 Ratio_correction_phase:REAL;  (* AV *)
	  Acceleration_correction_phase:REAL;  (* AA *)
	  
	  (* ===== registration ====*)
	  avec_registration:BOOL;
	  filtres_longueur_ON:BOOL;     // FL, FH, ZL, ZH 
	  Filtre_FL:REAL;
	  Filtre_FH:REAL;
	  Filtre_ZL:REAL;
	  Filtre_ZH:REAL;
	  
	  (* ====== Entrées sorties spéciales ======= *)
	  EntreeDeReference:BYTE := 3; // 0 = LOW, 1 = HIGH, 3=BE1, 4=BE1 invertiert,5=BE2, 6=BE2 invertiert,7=BE3, 8=BE3 invertiert,9=BE4, 10=BE4 invertiert,11=BE5, 12=BE5 invertiert,13=BE6, 14=BE6 invertiert,15=BE7, 16=BE7 invertiert,17=BE8, 18=BE8 invertiert,19=BE9, 20=BE9 invertiert,21=BE10, 22=BE10 invertiert,23=BE11, 24=BE11 invertiert,25=BE12, 26=BE12 invertiert,27=BE13, 28=BE13 invertiert, , 32=Bussteuersignal1, 33=Bussteuersignal2, 34=Bussteuersignal3, 35=Bussteuersignal4, 36=Bussteuersignal5
	  
	  
	  (* ====== Utilisation différentiel ======= *)
	  Utiliser_differentiel:BOOL;
	  
	  type_de_differentiel:BYTE;

(*	  
Pour définir l'axe en mode différentiel (L'axe a deux maitres : un via ML  l'autre via NL) il faut mettre le bit4 à 1
Pour choisir l'action des axes il faut choisir les bit5 & bit6 ainsi :    				  
LW 0001 0000  : 	ML + NL  		bit 5=0 ; bit6=0
LW 0111 0000 : 	ML - NL		bit 5=1 ; bit6=1
LW 0101 0000 : 	- ML - NL		bit 5=0 ; bit6=1
LW 0011 0000 : 	- ML + NL		bit 5=1 ; bit6=0
*)
	  
END_STRUCT


END_TYPE

// Status_axe
TYPE Status_axe :
	
STRUCT
		
	Loop_closed_PC:BOOL;
	Loop_open_MO:BOOL;
	Alignement_A_in_use:BOOL;                           // code 68
	Clutch_C_master_does_not_move:BOOL;    // code 66
	Clutch_C_master_move:BOOL;                      // code 67
	Interpolation_N_in_use:BOOL;
	Jog_VC_in_use:BOOL;
	move_MA_in_use:BOOL;
	Mapping_XM_in_use:BOOL;                           // code 2048
	Stop_ST_in_use:BOOL;
	Homing_IN_in_use:BOOL;
	
END_STRUCT



END_TYPE

// Utilitaire_axe
TYPE Utilitaire_axe :
	
STRUCT
		
	sMap_in_use: STRING := 'papier'; (* Nom came ex: 'CAME1'    Synchro linéaire en position  'LINEAR'  Synchro linéaire en  vitesse  'VITESSE' *)
	sMap_after: STRING := 'papier'; (* Nom came ex: 'CAME1'    Synchro linéaire en position  'LINEAR'  Synchro linéaire en  vitesse  'VITESSE' *)
	bMap_new:BOOL;
(*============== status homing ===============*)
	
	bhoming_done:BOOL;
	
	
END_STRUCT


END_TYPE

// GVL
{attribute 'qualified_only'}
VAR_GLOBAL
	OpModeStober :SINT;
	TargetAbsolutePosition:LREAL;
	Speed:LREAL;
	CapteurReference:BOOL;
	Position_ZC_Axe_1:LREAL;
	Modbus_1 : BOOL := 0;
	Modbus_2 : BOOL :=0;
	clrfault:BOOL;
END_VAR

// GVL_EtherCAT
{attribute 'qualified_only'}
VAR_GLOBAL
	EtherCATSlavesNumber:WORD;
	
	ListeEtherCATSlaves:ARRAY [0..100] OF ETCSLAVE_diag;
	
END_VAR

// MC_Pi
{attribute 'qualified_only'}
VAR_GLOBAL

AxesETC:ARRAY[1..100] OF axis_ref_sm3 ;

END_VAR

// var_infor
{attribute 'qualified_only'}
VAR_GLOBAL



info: ARRAY [1..1100] OF info_axe;



PLC_cycle_time:REAL; (* en sec *)

(*============== status maps ===============*)
	
bMaps_done:BOOL;

	
END_VAR

// Var_PMC
{attribute 'qualified_only'}
VAR_GLOBAL


(* Déclarer les axes sous la forme :

nom_descriptif_de_l_axe : udint := numero de l'axe; ( Numéro de l'axe est donné à titre indicatif, peu important, 
il servira d'index pour le stockage des paramètres dans les différents tableaux (PMC,SPEC_PMC_Util_PMC,...)

Exemple : 
Piston : udint := 1;

*)

Piston:UDINT:=1;
Virtuel:UDINT:=2;
Virtuel_1 : UDINT := 3;



PMC: ARRAY [1..1100] OF Parametres_axe;
Spec_PMC:  ARRAY [1..1100] OF specifiques_axe;
Util_PMC:  ARRAY [1..1100] OF Utilitaire_axe;
Status_PMC:  ARRAY [1..1100] OF Status_axe;
ListeNumSerieEthercat: ARRAY [1001..1100] OF udint;

NumeroDeSerieOk: ARRAY [1..1100] OF BOOL;
ListeAxesPrets: ARRAY [1..1100] OF BOOL;

Safety_relai_tempo:TIME:=T#3000MS;

retard_MO_PC:TIME:=T#600MS; (* Il faut attendre après avoir fait un MO pour relancer un PC sur PMCprotegoD *)
retard_PC_MO:TIME:=T#400MS; (* Il faut attendre après avoir fait un PC pour relancer un MO sur PMCprotegoD *)
Reset_fault:BOOL;

Utiliser_robot_gantry:BOOL;


bMap_OK:BOOL;   // génération des lois OK

Parameter_OK:BOOL; // Tous les paramètres variateurs et axes ont été chargés
//memoireNumSerieEthercat: ARRAY [1001..1100] OF udint := [9018034,9016089,442800005];

END_VAR

// Device/Application/PLC_PRG
PROGRAM PLC_PRG
VAR


	MC_Power_1: MC_Power;
	enable_virtuel: BOOL;
	mcpower1: BOOL;
	MC_MoveVelocity_1: MC_MoveVelocity;
	VC_virtuel: BOOL;
	MC_Stop_0: MC_Stop;
	MCSTOP: BOOL;
	MC_Reset_1: MC_Reset;
	activer_regulator: BOOL;
	Reset:bool;
	MC_Power_0: MC_Power;
	ActiverRegulateurAxe1: BOOL;
	EnableAxe1: BOOL;
	StatusAxe1: BOOL;
	MC_MoveVelocity_0: MC_MoveVelocity;
	VC_axe1: BOOL;
	VCActif: BOOL;
	VC_actif: BOOL;
	MC_Stop_1: MC_Stop;
	StopAxe1: BOOL;
	MC_Reset_0: MC_Reset;
	ResetAxe1: BOOL;
	MC_Jog_0: MC_Jog;
	JOGAvant: BOOL;
	JOGArriere: BOOL;
	MC_MoveAbsolute_0: MC_MoveAbsolute;
	MoveAbsolute: BOOL;
	MoveAbsoluteActif: BOOL;
	MoveAbsoluteFait: BOOL;
	MC_Home_0: MC_Home;
	Home: BOOL;
	SMC_Homing_0: SMC_Homing;
	MC_Home_1: MC_Home;
	ZC_Virtuel: BOOL;
	ZC_Axe1: BOOL;
	bRegulatorOnON: BOOL;
	MC_GearIn_0: MC_GearIn;
	XM: BOOL;
	AXIS_REF_ETC_STOEBER_SI6_SC6_0: AXIS_REF_ETC_STOEBER_SI6_SC6;
	MC_CamIn_0: MC_CamIn;
	CamIn: BOOL;
	MC_GearOut_0: MC_GearOut;
	GearOut: BOOL;
	MC_ReadActualPosition_0: MC_ReadActualPosition;
	Reset_virtuel: BOOL;
	NombreEsclavesEtherCAT_0: NombreEsclavesEtherCAT;
	LireNombreEsclavesEtherCAT: BOOL;
	SlaveType_0: SlaveType;
	SlaveType_1: SlaveType;
	fairesv: BOOL;
END_VAR

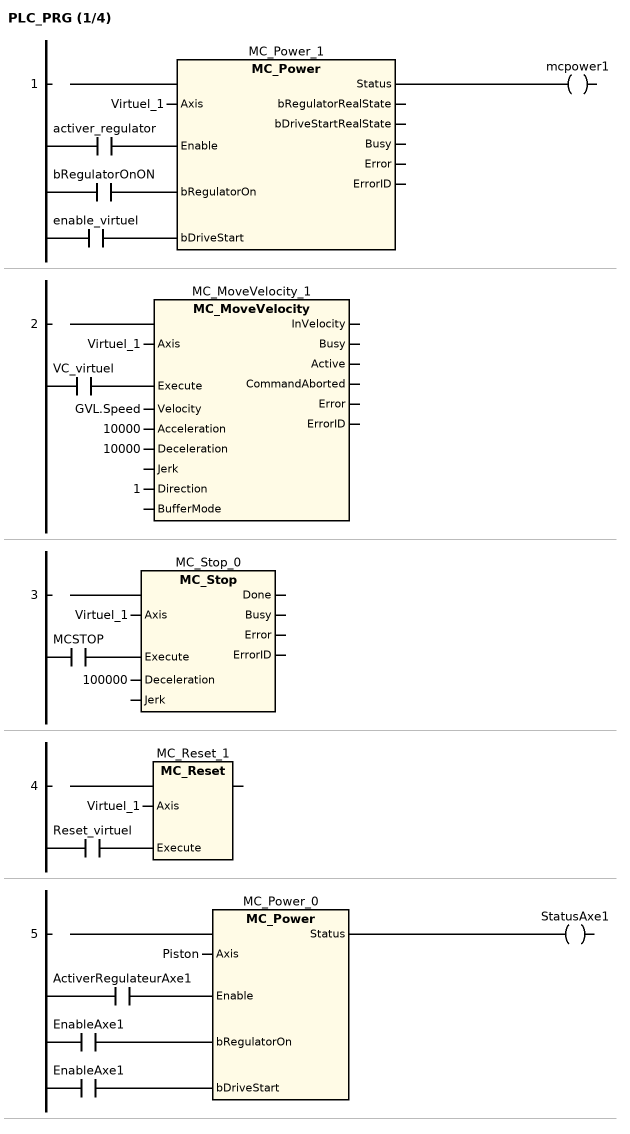
// NETWORK 1
MC_Power_1(
    Axis := Virtuel_1,
    Enable := activer_regulator,
    bRegulatorOn := bRegulatorOnON,
    bDriveStart := enable_virtuel); // MC_Power
mcpower1 := MC_Power_1.Status;

// NETWORK 2
MC_MoveVelocity_1(
    Axis := Virtuel_1,
    Execute := VC_virtuel,
    Velocity := GVL.Speed,
    Acceleration := 10000,
    Deceleration := 10000,
    Direction := 1); // MC_MoveVelocity

// NETWORK 3
MC_Stop_0(Axis := Virtuel_1, Execute := MCSTOP, Deceleration := 100000); // MC_Stop

// NETWORK 4
MC_Reset_1(Axis := Virtuel_1, Execute := Reset_virtuel); // MC_Reset

// NETWORK 5
MC_Power_0(
    Axis := Piston,
    Enable := ActiverRegulateurAxe1,
    bRegulatorOn := EnableAxe1,
    bDriveStart := EnableAxe1); // MC_Power
StatusAxe1 := MC_Power_0.Status;

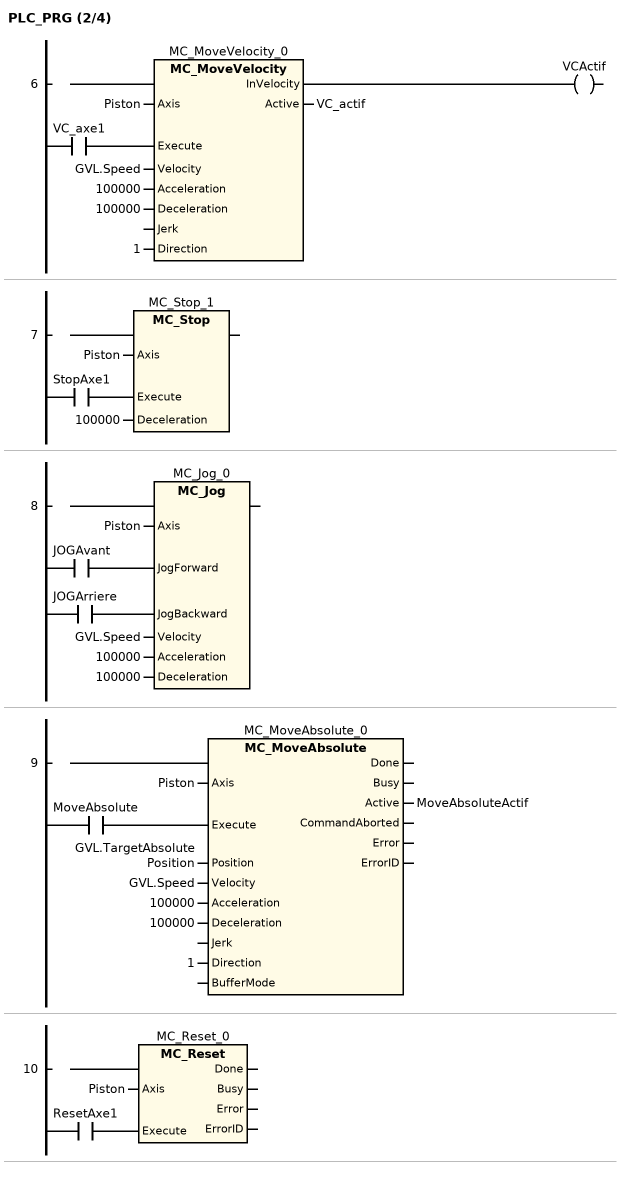
// NETWORK 6
MC_MoveVelocity_0(
    Axis := Piston,
    Execute := VC_axe1,
    Velocity := GVL.Speed,
    Acceleration := 100000,
    Deceleration := 100000,
    Direction := 1,
    Active => VC_actif); // MC_MoveVelocity
VCActif := MC_MoveVelocity_0.InVelocity;

// NETWORK 7
MC_Stop_1(Axis := Piston, Execute := StopAxe1, Deceleration := 100000); // MC_Stop

// NETWORK 8
MC_Jog_0(
    Axis := Piston,
    JogForward := JOGAvant,
    JogBackward := JOGArriere,
    Velocity := GVL.Speed,
    Acceleration := 100000,
    Deceleration := 100000); // MC_Jog

// NETWORK 9
MC_MoveAbsolute_0(
    Axis := Piston,
    Execute := MoveAbsolute,
    Position := GVL.TargetAbsolutePosition,
    Velocity := GVL.Speed,
    Acceleration := 100000,
    Deceleration := 100000,
    Direction := 1,
    Active => MoveAbsoluteActif); // MC_MoveAbsolute

// NETWORK 10
MC_Reset_0(Axis := Piston, Execute := ResetAxe1); // MC_Reset

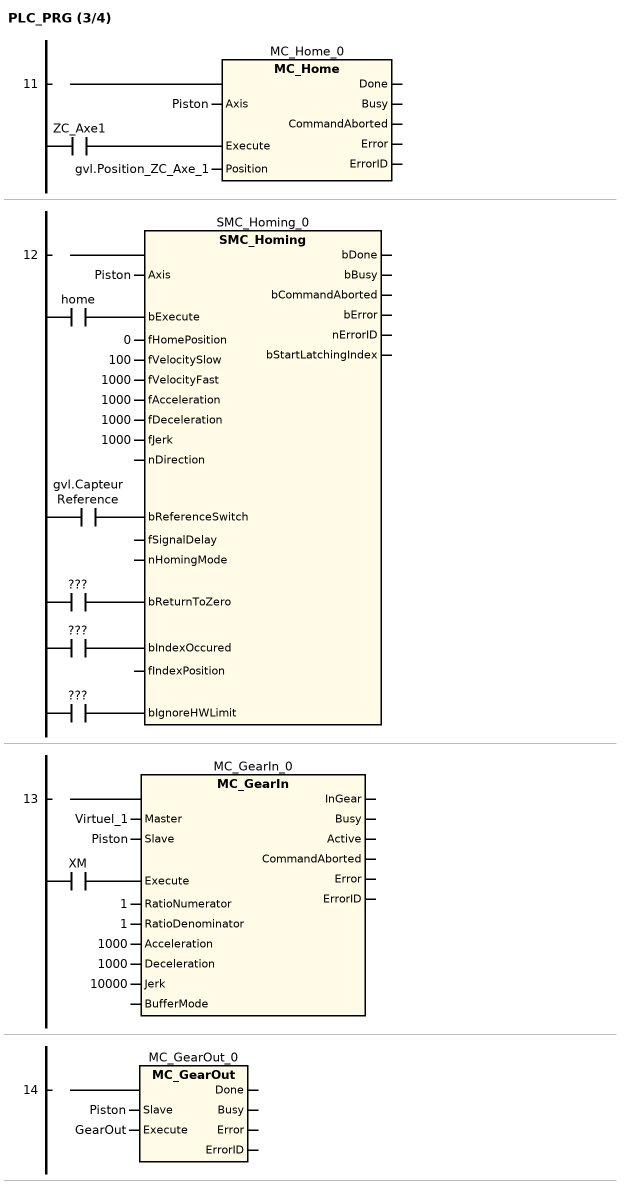
// NETWORK 11
MC_Home_0(Axis := Piston, Execute := ZC_Axe1, Position := gvl.Position_ZC_Axe_1); // MC_Home

// NETWORK 12
SMC_Homing_0(
    Axis := Piston,
    bExecute := home,
    fHomePosition := 0,
    fVelocitySlow := 100,
    fVelocityFast := 1000,
    fAcceleration := 1000,
    fDeceleration := 1000,
    fJerk := 1000,
    bReferenceSwitch := gvl.CapteurReference); // SMC_Homing

// NETWORK 13
MC_GearIn_0(
    Master := Virtuel_1,
    Slave := Piston,
    Execute := XM,
    RatioNumerator := 1,
    RatioDenominator := 1,
    Acceleration := 1000,
    Deceleration := 1000,
    Jerk := 10000); // MC_GearIn

// NETWORK 14
MC_GearOut_0(Slave := Piston, Execute := GearOut); // MC_GearOut

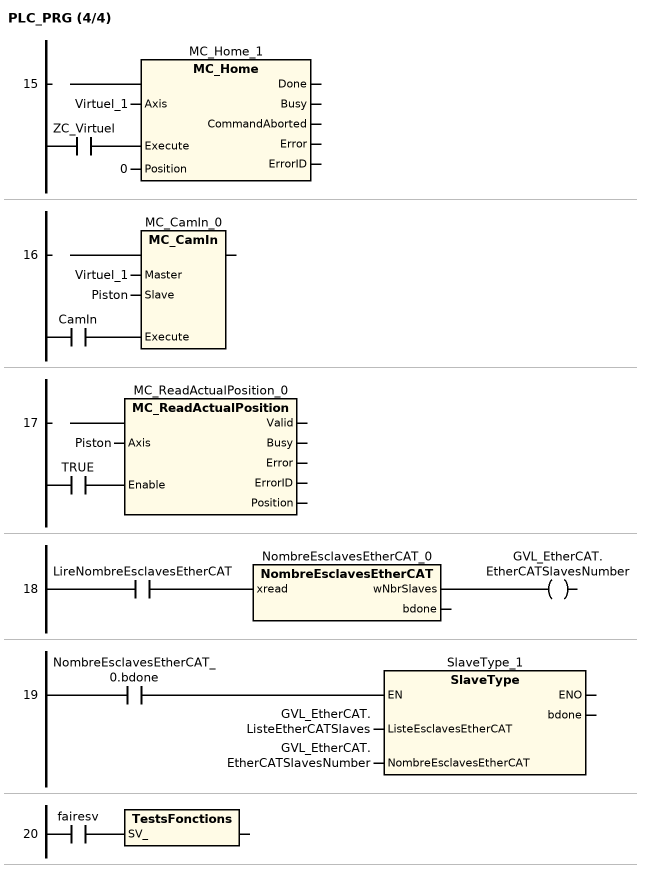
// NETWORK 15
MC_Home_1(Axis := Virtuel_1, Execute := ZC_Virtuel, Position := 0); // MC_Home

// NETWORK 16
MC_CamIn_0(Master := Virtuel_1, Slave := Piston, Execute := CamIn); // MC_CamIn

// NETWORK 17
MC_ReadActualPosition_0(Axis := Piston, Enable := TRUE); // MC_ReadActualPosition

// NETWORK 18
NombreEsclavesEtherCAT_0(xread := LireNombreEsclavesEtherCAT); // NombreEsclavesEtherCAT
GVL_EtherCAT.EtherCATSlavesNumber := NombreEsclavesEtherCAT_0.wNbrSlaves;

// NETWORK 19
IF NombreEsclavesEtherCAT_0.bdone THEN
    SlaveType_1(ListeEsclavesEtherCAT := GVL_EtherCAT.ListeEtherCATSlaves, NombreEsclavesEtherCAT := GVL_EtherCAT.EtherCATSlavesNumber); // SlaveType
END_IF

// NETWORK 20
TestsFonctions(SV_ := fairesv);

END_PROGRAM

// EtherCAT/NombreEsclavesEtherCAT
FUNCTION_BLOCK NombreEsclavesEtherCAT
VAR_INPUT
	xread:BOOL;
END_VAR
VAR_OUTPUT
	wNbrSlaves:WORD;
	bdone:bool;
END_VAR
VAR
	readnbr : ReadNbrSlaves;
	pointeur:POINTER TO INT ;
	ID:int;
END_VAR

IF xRead THEN
   readnbr.usiCom := DWORD_TO_USINT(EtherCAT_Master_Softmotion.InstanceNumber);
   readnbr(xExecute := TRUE, udiTimeOut := 1000);
   IF readnbr.xDone THEN
      xRead := FALSE;
      wNbrSlaves := readnbr.wNumberSlaves;
      readnbr(xExecute := FALSE);
	  bdone:=TRUE;
	  pointeur:= EtherCAT_Master_Softmotion.FirstSlave;

    END_IF
 END_IF

END_FUNCTION_BLOCK

// EtherCAT/SlaveType
//Détermine le type d'esclave EtherCAT
//Exemples : Variateur | Codeur | Bloc d'E/S

FUNCTION_BLOCK SlaveType
VAR_INPUT
	ListeEsclavesEtherCAT: ARRAY [0..100] OF ETCSLAVE_diag;
	
	NombreEsclavesEtherCAT:INT;
END_VAR
VAR_OUTPUT
	bdone:BOOL;
END_VAR
VAR
	TypeEsclaveEtherCAT: ARRAY [0..100] OF DWORD;
	index:INT:=0;
END_VAR

FOR index:=0 TO NombreEsclavesEtherCAT BY 1 DO 
	TypeEsclaveEtherCAT[index]:= ListeEsclavesEtherCAT[index].ProductID;
	IF index>NombreEsclavesEtherCAT THEN
		
		bdone:=TRUE;
		RETURN;
	END_IF
END_FOR

END_FUNCTION_BLOCK

// TestsFonctions
PROGRAM TestsFonctions
VAR_INPUT
	SV_:BOOL;
END_VAR

END_PROGRAM

// POU
PROGRAM POU
VAR
	
	Lancer_gestionaxes: BOOL;
	MC_CamIn_0: SM3_Basic.MC_CamIn;
	CamIn: BOOL;
	passagevirtuel: BOOL;
	reinitdrive: BOOL;
	SMC3_ReinitDrive_1: SM3_Basic.SMC3_ReinitDrive;
	rien: BOOL;
	PasserenVirtuel: BOOL;
	MC_Reset_0: SM3_Basic.MC_Reset;
	Reset_: BOOL;
	SMC_CheckAxisCommunication_0: SM3_Basic.SMC_CheckAxisCommunication;
	Check: BOOL;
END_VAR

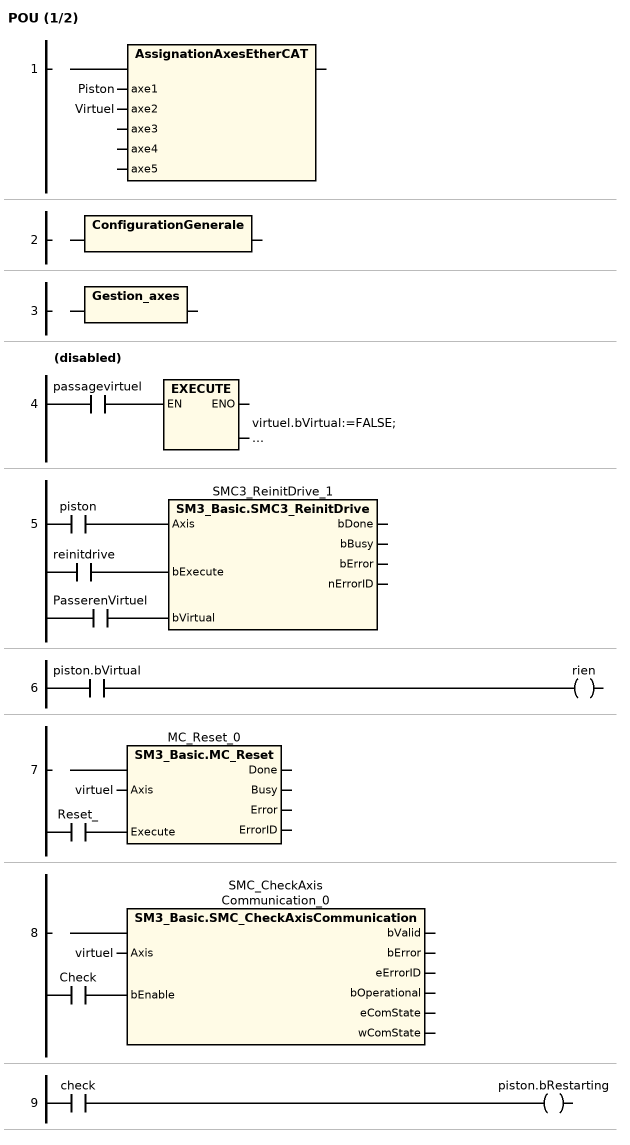
// NETWORK 1
AssignationAxesEtherCAT(axe1 := Piston, axe2 := Virtuel);

// NETWORK 2
ConfigurationGenerale();

// NETWORK 3
Gestion_axes();

// NETWORK 4 (disabled)
// IF passagevirtuel THEN virtuel.bVirtual:=FALSE; END_IF

// NETWORK 5
SMC3_ReinitDrive_1(Axis := piston, bExecute := reinitdrive, bVirtual := PasserenVirtuel); // SM3_Basic.SMC3_ReinitDrive

// NETWORK 6
rien := piston.bVirtual;

// NETWORK 7
MC_Reset_0(Axis := virtuel, Execute := Reset_); // SM3_Basic.MC_Reset

// NETWORK 8
SMC_CheckAxisCommunication_0(Axis := virtuel, bEnable := Check); // SM3_Basic.SMC_CheckAxisCommunication

// NETWORK 9
piston.bRestarting := check;

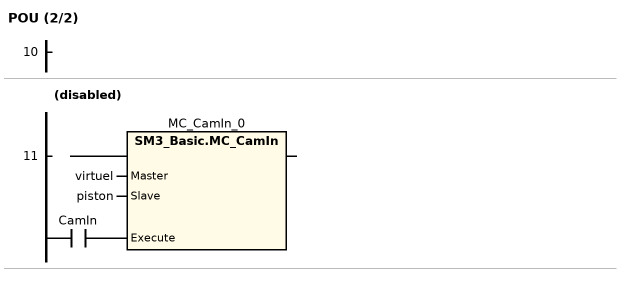
// NETWORK 10

// NETWORK 11 (disabled)
// MC_CamIn_0(Master := virtuel, Slave := piston, Execute := CamIn); // SM3_Basic.MC_CamIn

END_PROGRAM

// AssignationAxesEtherCAT
PROGRAM AssignationAxesEtherCAT
VAR_INPUT
	axe1:axis_ref_sm3;
	axe2:axis_ref_sm3;
	axe3:axis_ref_sm3;
	axe4:axis_ref_sm3;
	axe5:axis_ref_sm3;
END_VAR

mc_pi.AxesETC[1]:=axe1;
mc_pi.AxesETC[2]:=axe2;
mc_pi.AxesETC[3]:=axe3;
mc_pi.AxesETC[4]:=axe4;
mc_pi.AxesETC[5]:=axe5;

END_PROGRAM

// ConfigurationGenerale
PROGRAM ConfigurationGenerale
VAR
	
END_VAR

(*================= Axes réels EtherCAT ====================*)

(*==================================================================================================================================================================*)

var_PMC.PMC[VAR_PMC.piston].sNom:='Piston';
var_PMC.PMC[VAR_PMC.piston].sMoteur:= 'EZ302OCst';
var_PMC.PMC[VAR_PMC.piston].sTypeDeVariateur:= 'SC6';
var_pmc.PMC[VAR_PMC.piston].sChoixAxe:='A';
var_pmc.PMC[VAR_PMC.piston].dwAdresseEtherCAT:=1001;
var_PMC.PMC[VAR_PMC.piston].sNomMaitre:='';
var_PMC.PMC[VAR_PMC.piston].sNomMaitreDifferentiel:='';
var_PMC.PMC[VAR_PMC.piston].diCycle:=22220000; 									(* SB *)
var_PMC.PMC[VAR_PMC.piston].rEchelle:=100;
var_PMC.PMC[VAR_PMC.piston].diContrainte_Mvt:=20000;
var_PMC.PMC[VAR_PMC.piston].diContrainte_Mvt_neg:=20000;
var_PMC.PMC[VAR_PMC.piston].bsens:=0;												(* CW *)
var_PMC.PMC[VAR_PMC.piston].rTolerance_poursuite_Maxi:=2;  			(* SE *)

	(* ===== mouvement =====*)
	
var_PMC.PMC[VAR_PMC.piston].rVitesse:=180;											(* SV *)
var_PMC.PMC[VAR_PMC.piston].racceleration:=10000;							(* SA *)
var_PMC.PMC[VAR_PMC.piston].rdecceleration:=10000;                       (* DC *)
var_PMC.PMC[VAR_PMC.piston].rdecceleration_urgence:=20000;  		(* XA *)
var_PMC.PMC[VAR_PMC.piston].rPosArret:=0;												(* ST position ou MA position *)
(*============== registration ===============*)
var_PMC.PMC[VAR_PMC.piston].rCorrection_Registration:=2;    			(* SR *)
var_PMC.PMC[VAR_PMC.piston].rfiltre_Registration:=2;    						(* FR *)
var_PMC.PMC[VAR_PMC.piston].usicontrole_Registration:=2;    			(* RT *)
var_PMC.PMC[VAR_PMC.piston].rPosCapteur:=0;    								(* RF *)
var_PMC.Spec_PMC[VAR_PMC.piston].avec_registration:=TRUE;
var_PMC.Spec_PMC[VAR_PMC.piston].EntreeDeReference:=3; // 0 = LOW, 1 = HIGH, 3=BE1, 4=BE1 invertiert,5=BE2, 6=BE2 invertiert,7=BE3, 8=BE3 invertiert,9=BE4, 10=BE4 invertiert,11=BE5, 12=BE5 invertiert,13=BE6, 14=BE6 invertiert,15=BE7, 16=BE7 invertiert,17=BE8, 18=BE8 invertiert,19=BE9, 20=BE9 invertiert,21=BE10, 22=BE10 invertiert,23=BE11, 24=BE11 invertiert,25=BE12, 26=BE12 invertiert,27=BE13, 28=BE13 invertiert, , 32=Bussteuersignal1, 33=Bussteuersignal2, 34=Bussteuersignal3, 35=Bussteuersignal4, 36=Bussteuersignal5
(*============= embrayage  synchronisation ===*)
var_PMC.PMC[VAR_PMC.piston].rFenetre_Embrayage:=2;    					(* CI *)
var_PMC.PMC[VAR_PMC.piston].rdistance_Embrayage:=20;    				(* CL  ou CT*)
var_PMC.PMC[VAR_PMC.piston].rphase_maitre:=2;    											(* MB*)
var_PMC.PMC[VAR_PMC.piston].stype_embrayage:='ALIGNEMENT_COURT';
var_PMC.PMC[VAR_PMC.piston].sLoi_MVT:='MAP';    				

var_PMC.PMC[VAR_PMC.piston].Gain_vitesse:=0.15;    							(* GV *)
var_PMC.PMC[VAR_PMC.piston].Tension_secteur:=2;   
var_PMC.PMC[VAR_PMC.piston].Mode_Asservissement:=24;    	 		(* FS *)
var_PMC.PMC[VAR_PMC.piston].Frein:=FALSE;    													(* MBRAKE *)

(* specifique *)
var_PMC.Spec_PMC[VAR_PMC.piston].Multiplication_points_codeur:=0;    (* MS *)
var_PMC.Spec_PMC[VAR_PMC.piston].Filtre_codeur:=0;  (* PT *)		
				
var_PMC.Spec_PMC[VAR_PMC.piston].Ratio_correction_phase:=20;  (* AV *)
var_PMC.Spec_PMC[VAR_PMC.piston].Acceleration_correction_phase:=var_PMC.PMC[VAR_PMC.piston].rAcceleration;  (* AA *)

(*==================================================================================================================================================================*)

(*==================================================================================================================================================================*)

var_PMC.PMC[VAR_PMC.virtuel].sNom:='Virtuel';
var_PMC.PMC[VAR_PMC.virtuel].sMoteur:= 'EZ302OCst';
var_PMC.PMC[VAR_PMC.virtuel].sTypeDeVariateur:= '';
var_pmc.PMC[VAR_PMC.virtuel].sChoixAxe:='';
var_pmc.PMC[VAR_PMC.virtuel].dwAdresseEtherCAT:=1002;
var_PMC.PMC[VAR_PMC.virtuel].sNomMaitre:='';
var_PMC.PMC[VAR_PMC.virtuel].sNomMaitreDifferentiel:='';
var_PMC.PMC[VAR_PMC.virtuel].diCycle:=22220000; 									(* SB *)
var_PMC.PMC[VAR_PMC.virtuel].rEchelle:=100;
var_PMC.PMC[VAR_PMC.virtuel].diContrainte_Mvt:=20000;
var_PMC.PMC[VAR_PMC.virtuel].diContrainte_Mvt_neg:=20000;
var_PMC.PMC[VAR_PMC.virtuel].bsens:=0;												(* CW *)
var_PMC.PMC[VAR_PMC.virtuel].rTolerance_poursuite_Maxi:=2;  			(* SE *)
	(* ===== mouvement =====*)
	
var_PMC.PMC[VAR_PMC.virtuel].rVitesse:=180;											(* SV *)
var_PMC.PMC[VAR_PMC.virtuel].racceleration:=10000;							(* SA *)
var_PMC.PMC[VAR_PMC.virtuel].rdecceleration:=10000;                       (* DC *)
var_PMC.PMC[VAR_PMC.virtuel].rdecceleration_urgence:=20000;  		(* XA *)
var_PMC.PMC[VAR_PMC.virtuel].rPosArret:=0;												(* ST position ou MA position *)
(*============== registration ===============*)
var_PMC.PMC[VAR_PMC.virtuel].rCorrection_Registration:=2;    			(* SR *)
var_PMC.PMC[VAR_PMC.virtuel].rfiltre_Registration:=2;    						(* FR *)
var_PMC.PMC[VAR_PMC.virtuel].usicontrole_Registration:=2;    			(* RT *)
var_PMC.PMC[VAR_PMC.virtuel].rPosCapteur:=0;    								(* RF *)
var_PMC.Spec_PMC[VAR_PMC.virtuel].avec_registration:=TRUE;
var_PMC.Spec_PMC[VAR_PMC.virtuel].EntreeDeReference:=3; // 0 = LOW, 1 = HIGH, 3=BE1, 4=BE1 invertiert,5=BE2, 6=BE2 invertiert,7=BE3, 8=BE3 invertiert,9=BE4, 10=BE4 invertiert,11=BE5, 12=BE5 invertiert,13=BE6, 14=BE6 invertiert,15=BE7, 16=BE7 invertiert,17=BE8, 18=BE8 invertiert,19=BE9, 20=BE9 invertiert,21=BE10, 22=BE10 invertiert,23=BE11, 24=BE11 invertiert,25=BE12, 26=BE12 invertiert,27=BE13, 28=BE13 invertiert, , 32=Bussteuersignal1, 33=Bussteuersignal2, 34=Bussteuersignal3, 35=Bussteuersignal4, 36=Bussteuersignal5
(*============= embrayage  synchronisation ===*)
var_PMC.PMC[VAR_PMC.virtuel].rFenetre_Embrayage:=2;    					(* CI *)
var_PMC.PMC[VAR_PMC.virtuel].rdistance_Embrayage:=20;    				(* CL  ou CT*)
var_PMC.PMC[VAR_PMC.virtuel].rphase_maitre:=2;    											(* MB*)
var_PMC.PMC[VAR_PMC.virtuel].stype_embrayage:='ALIGNEMENT_COURT';
var_PMC.PMC[VAR_PMC.virtuel].sLoi_MVT:='MAP';    				

var_PMC.PMC[VAR_PMC.virtuel].Gain_vitesse:=0.15;    							(* GV *)
var_PMC.PMC[VAR_PMC.virtuel].Tension_secteur:=2;   
var_PMC.PMC[VAR_PMC.virtuel].Mode_Asservissement:=24;    	 		(* FS *)
var_PMC.PMC[VAR_PMC.virtuel].Frein:=FALSE;    													(* MBRAKE *)

(* specifique *)
var_PMC.Spec_PMC[VAR_PMC.virtuel].Multiplication_points_codeur:=0;    (* MS *)
var_PMC.Spec_PMC[VAR_PMC.virtuel].Filtre_codeur:=0;  (* PT *)		
				
var_PMC.Spec_PMC[VAR_PMC.virtuel].Ratio_correction_phase:=20;  (* AV *)
var_PMC.Spec_PMC[VAR_PMC.virtuel].Acceleration_correction_phase:=var_PMC.PMC[VAR_PMC.virtuel].rAcceleration;  (* AA *)

END_PROGRAM

// Gestion axes/Gestion_axes
PROGRAM Gestion_axes
VAR
	Gr_Piston: Gr_Axe;
	Gr_virtuel: Gr_Axe;
END_VAR

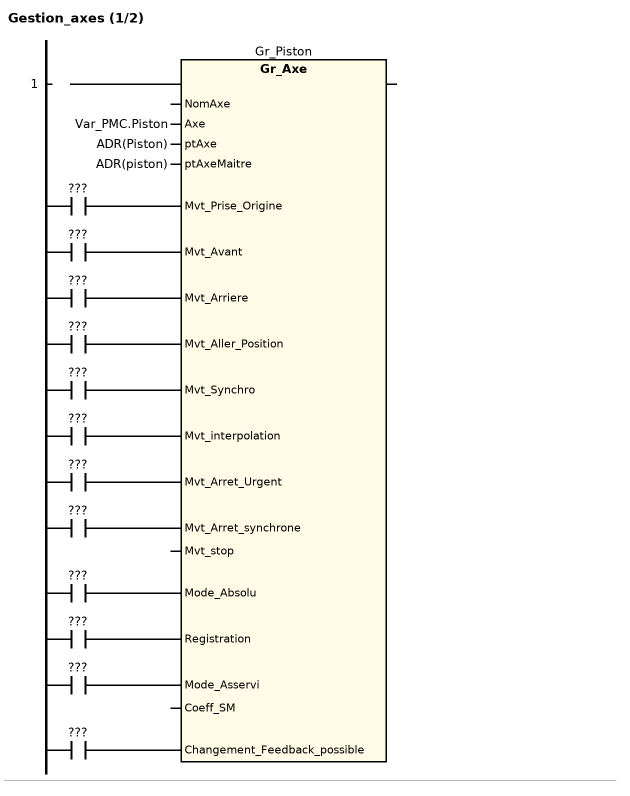
// NETWORK 1
Gr_Piston(Axe := Var_PMC.Piston, ptAxe := ADR(Piston), ptAxeMaitre := ADR(piston)); // Gr_Axe

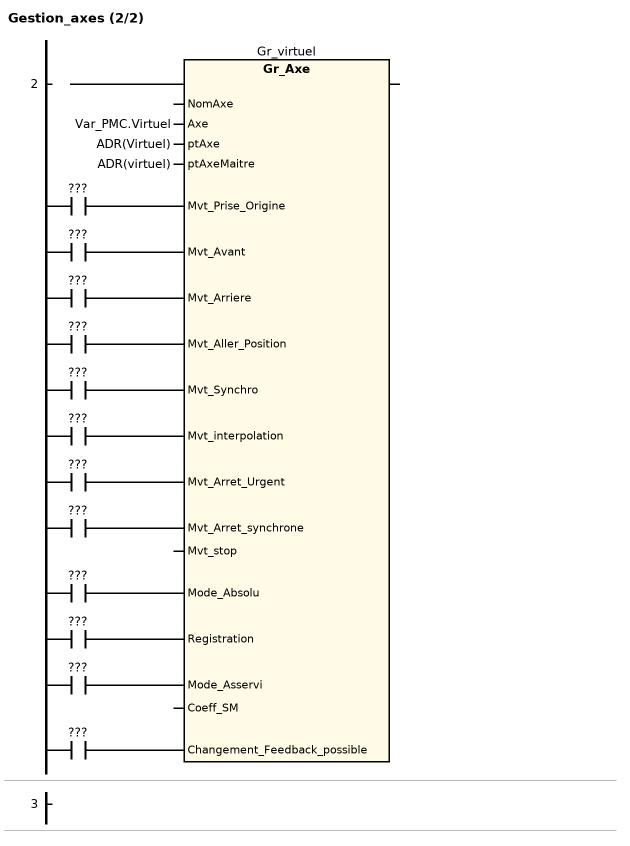
// NETWORK 2
Gr_virtuel(Axe := Var_PMC.Virtuel, ptAxe := ADR(Virtuel), ptAxeMaitre := ADR(virtuel)); // Gr_Axe

// NETWORK 3

END_PROGRAM

// Gestion axes/Gr_Axe
FUNCTION_BLOCK Gr_Axe
VAR_INPUT
	NomAxe:STRING;
	Axe:UDINT;
	ptAxe: POINTER TO axis_ref_sm3; //Entrer le nom de l'axe comme défini dans l'architecure matérielle. 
	ptAxeMaitre: POINTER TO axis_ref_sm3; // Entrer le nom de l'axe comme défini dans l'architecture matérielle. Si pas de synchro (donc pas de maître), entrer le nom de l'axe lui même
	MasterAxis: POINTER TO axis_ref_sm3;
	PointeurRien : POINTER TO axis_ref_sm3;
	//structAxe:axis_ref_sm3;
	//StAxe:AXIS_REF_ETC_STOEBER_SI6_SC6;
	Mvt_Prise_Origine:BOOL; (* Mouvement  prise origine *)
	Mvt_Avant: BOOL; (* Mouvement indépendant en Avant *)
	Mvt_Arriere: BOOL; (* Mouvement indépendant en Arriére *)
	Mvt_Aller_Position: BOOL; (* Aller à la position Cible ( Variable PosArret ) *)
	Mvt_Synchro: BOOL; (* Demande de XM *)
	Mvt_interpolation: BOOL; (* Axis Control *)
	Mvt_Arret_Urgent: BOOL; (* Demande Arret Urgent *)
	Mvt_Arret_synchrone: BOOL; (* demande Stop en position sur loi de mvt en cours *)
	Mvt_stop:BOOL; (*Stop*)
	//Autre_mvt_demande:bool; (*Par exemple un mouvement relatif *)
	Mode_Absolu: BOOL; (* Initialisation obligatoire ou pas *)
	Registration:BOOL; (*Avec ou sans registration*)
	Mode_Asservi: BOOL;
	Coeff_SM: REAL;
	Utiliser_boucle_codeur_externe:BOOL;
	Changement_Feedback_possible:BOOL;
	tactile: BOOL;
	
	
END_VAR
VAR_OUTPUT
END_VAR
VAR
	
	sAxe:STRING:=concat('VAR_PMC.',NomAxe);
	Activation_homing: BOOL;

	Activation_Jog: BOOL;
	
	Activation_Mapping: BOOL;
	
	
	Activation_MoveToPosition: BOOL;
	bCommon_Stop: BOOL;
	
	
	
	SetChannelParametersDone: BOOL;
	Dans_homing: BOOL;
	SMC_Homing_1: SMC_Homing;
	SMC_Homing_0: SMC_Homing;
	rien: BOOL;
	Activation_mvt: BOOL;
	
	MC_Jog_0: MC_Jog;
	MC_GearIn_0: MC_GearIn;
	MC_GearInPos_0: MC_GearInPos;
	MC_CamIn_0: MC_CamIn;
	AxisState: MC_ReadStatus;
	MC_Stop_0: MC_Stop;
	MC_Power_0: MC_Power;
	MC_Halt_0: MC_Halt;
	MC_MoveAbsolute_0: MC_MoveAbsolute;
	MC_Power_Off: MC_Power;
	MC_Power_on: MC_Power;
	MC_Reset_0: MC_Reset;
	MC_Stop_1: MC_Stop;
	resetErreur: BOOL;
	MC_Stop_2: MC_Stop;
	AxisDisabled: BOOL;
	AxisErrorStop: BOOL;
	AxisStopping: BOOL;
	AxisStandstill: BOOL;
	AxisDiscreteMotion: BOOL;
	AxisContinuousMotion: BOOL;
	AxisSynchronizedMotion: BOOL;
	AxisHoming: BOOL;
	AxisConstantVelocity: BOOL;
	AxisAccelerating: BOOL;
	AxisDecelerating: BOOL;
	SMC_ReadFBError_0: SMC_ReadFBError;
	compteur: INT;
	comptage: BOOL;
	MC_Home_0: MC_Home;
	MC_Home_1: MC_Home;
	MC_MoveVelocity_0: MC_MoveVelocity;
	forcer_passage: BOOL;
	MC_MoveAbsolute_1: MC_MoveAbsolute;
	MC_Jog_1: MC_Jog;
	MC_MoveAbsolute_2: MC_MoveAbsolute;
	fin_jog: BOOL;
	fin_homing: BOOL;
	Fin_Jog_immediat: BOOL;
	fin_move_stop_position: BOOL;
	Fin_liaison: BOOL;
	ajeh: BOOL;
	Fin_liaison_immediat: BOOL;
	Fin_stop: BOOL;
	Position_atteinte_0: Position_atteinte;
	PositionAtteinte: BOOL;
	fabien: BOOL;
	MC_GearIn_1: MC_GearIn;
	Camin: BOOL;
	Mc_GearIn_2: MC_gearIn;
	LecturePositionMaitre: SM3_Basic.MC_ReadActualPosition;
END_VAR

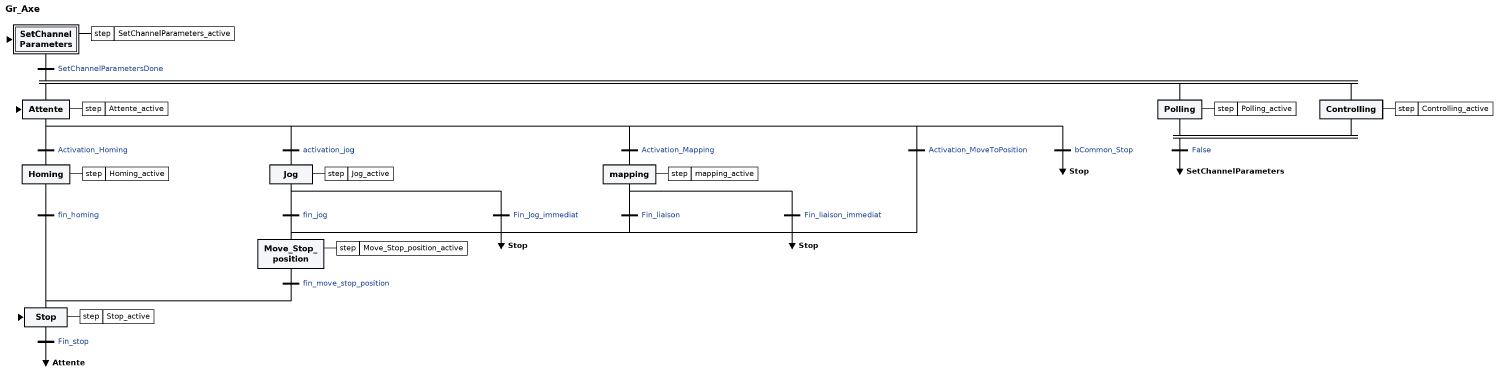
INITIAL_STEP SetChannelParameters:
    SetChannelParameters_active(N);  // step action
END_STEP
TRANSITION FROM SetChannelParameters TO (Attente, Polling, Controlling)
    := SetChannelParametersDone;
END_TRANSITION
STEP Attente:
    Attente_active(N);  // step action
END_STEP
STEP Polling:
    Polling_active(N);  // step action
END_STEP
STEP Controlling:
    Controlling_active(N);  // step action
END_STEP
TRANSITION FROM (Polling, Controlling) TO SetChannelParameters
    := False;
END_TRANSITION
TRANSITION FROM Attente TO Homing
    := Activation_Homing;
END_TRANSITION
STEP Homing:
    Homing_active(N);  // step action
END_STEP
TRANSITION FROM Homing TO Stop
    := fin_homing;
END_TRANSITION
TRANSITION FROM Attente TO Jog
    := activation_jog;
END_TRANSITION
STEP Jog:
    Jog_active(N);  // step action
END_STEP
TRANSITION FROM Jog TO Move_Stop_position
    := fin_jog;
END_TRANSITION
TRANSITION FROM Jog TO Stop
    := Fin_Jog_immediat;
END_TRANSITION
TRANSITION FROM Attente TO mapping
    := Activation_Mapping;
END_TRANSITION
STEP mapping:
    mapping_active(N);  // step action
END_STEP
TRANSITION FROM mapping TO Move_Stop_position
    := Fin_liaison;
END_TRANSITION
TRANSITION FROM mapping TO Stop
    := Fin_liaison_immediat;
END_TRANSITION
TRANSITION FROM Attente TO Move_Stop_position
    := Activation_MoveToPosition;
END_TRANSITION
STEP Move_Stop_position:
    Move_Stop_position_active(N);  // step action
END_STEP
TRANSITION FROM Move_Stop_position TO Stop
    := fin_move_stop_position;
END_TRANSITION
TRANSITION FROM Attente TO Stop
    := bCommon_Stop;
END_TRANSITION
STEP Stop:
    Stop_active(N);  // step action
END_STEP
TRANSITION FROM Stop TO Attente
    := Fin_stop;
END_TRANSITION

ACTION Attente_active:
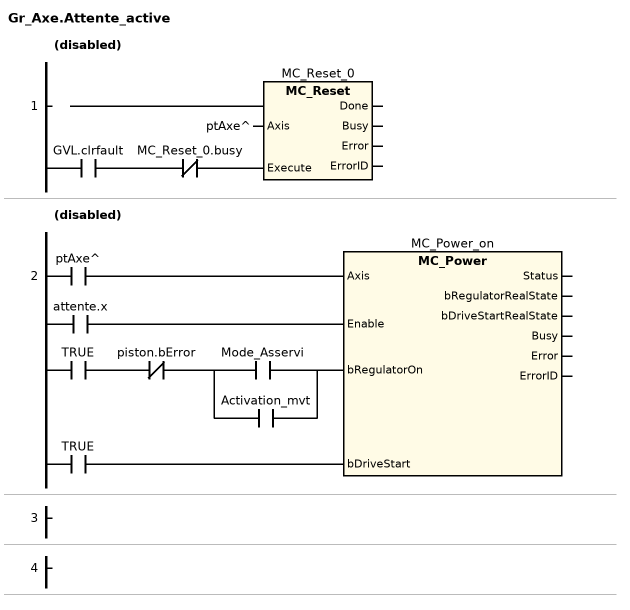
// NETWORK 1 (disabled)
// MC_Reset_0(Axis := ptAxe^, Execute := GVL.clrfault AND NOT MC_Reset_0.busy); // MC_Reset

// NETWORK 2 (disabled)
// MC_Power_on(
//     Axis := ptAxe^,
//     Enable := attente.x,
//     bRegulatorOn := TRUE AND NOT piston.bError AND (Mode_Asservi OR Activation_mvt),
//     bDriveStart := TRUE); // MC_Power

// NETWORK 3

// NETWORK 4
END_ACTION

ACTION Controlling_active:
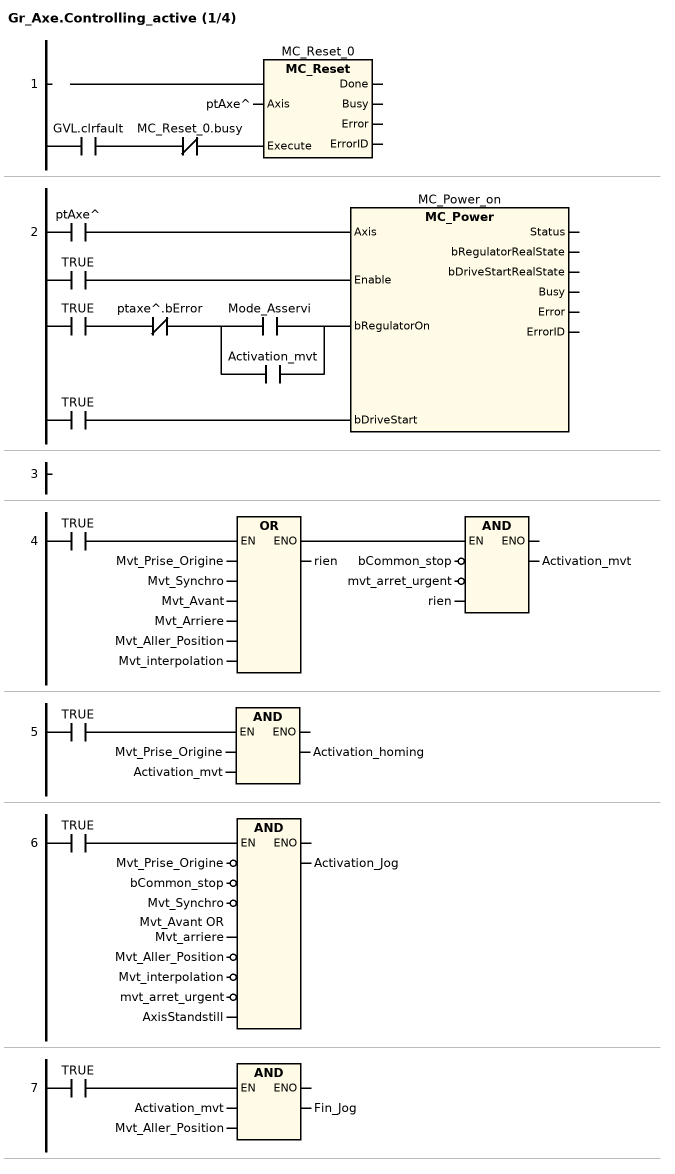
// NETWORK 1
MC_Reset_0(Axis := ptAxe^, Execute := GVL.clrfault AND NOT MC_Reset_0.busy); // MC_Reset

// NETWORK 2
MC_Power_on(
    Axis := ptAxe^,
    Enable := TRUE,
    bRegulatorOn := TRUE AND NOT ptaxe^.bError AND (Mode_Asservi OR Activation_mvt),
    bDriveStart := TRUE); // MC_Power

// NETWORK 3

// NETWORK 4
rien := Mvt_Prise_Origine OR Mvt_Synchro OR Mvt_Avant OR Mvt_Arriere OR Mvt_Aller_Position OR Mvt_interpolation;
Activation_mvt := NOT bCommon_stop AND NOT mvt_arret_urgent AND rien;

// NETWORK 5
Activation_homing := Mvt_Prise_Origine AND Activation_mvt;

// NETWORK 6
Activation_Jog := NOT Mvt_Prise_Origine AND NOT bCommon_stop AND NOT Mvt_Synchro AND (Mvt_Avant OR Mvt_arriere) AND NOT Mvt_Aller_Position AND NOT Mvt_interpolation AND NOT mvt_arret_urgent AND AxisStandstill;

// NETWORK 7
Fin_Jog := Activation_mvt AND Mvt_Aller_Position;

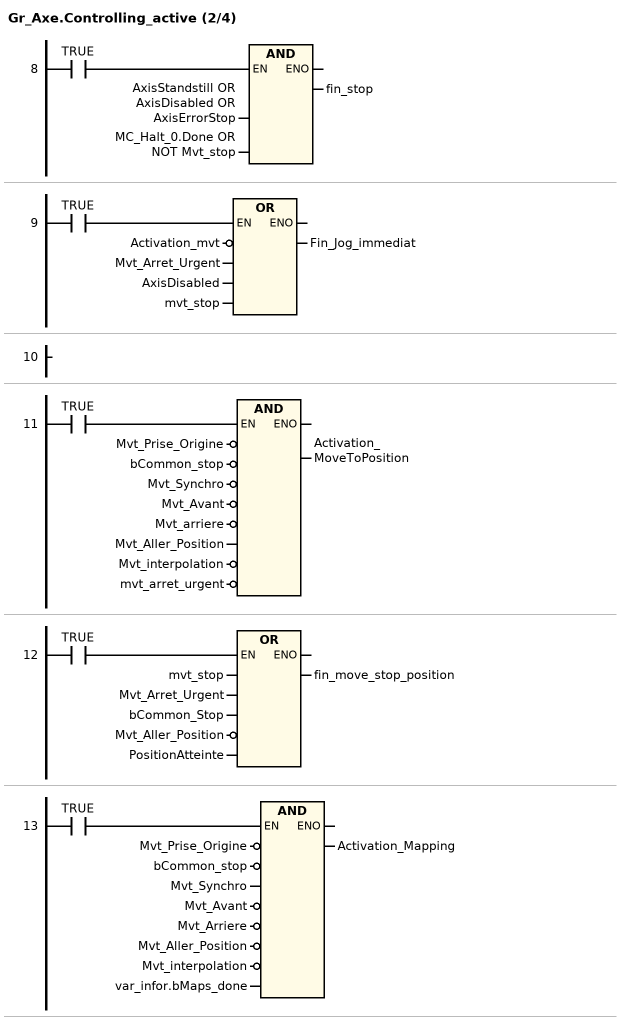
// NETWORK 8
fin_stop := (AxisStandstill OR AxisDisabled OR AxisErrorStop) AND (MC_Halt_0.Done OR NOT Mvt_stop);

// NETWORK 9
Fin_Jog_immediat := NOT Activation_mvt OR Mvt_Arret_Urgent OR AxisDisabled OR mvt_stop;

// NETWORK 10

// NETWORK 11
Activation_MoveToPosition := NOT Mvt_Prise_Origine AND NOT bCommon_stop AND NOT Mvt_Synchro AND NOT Mvt_Avant AND NOT Mvt_arriere AND Mvt_Aller_Position AND NOT Mvt_interpolation AND NOT mvt_arret_urgent;

// NETWORK 12
fin_move_stop_position := mvt_stop OR Mvt_Arret_Urgent OR bCommon_Stop OR NOT Mvt_Aller_Position OR PositionAtteinte;

// NETWORK 13
Activation_Mapping := NOT Mvt_Prise_Origine AND NOT bCommon_stop AND Mvt_Synchro AND NOT Mvt_Avant AND NOT Mvt_Arriere AND NOT Mvt_Aller_Position AND NOT Mvt_interpolation AND var_infor.bMaps_done;

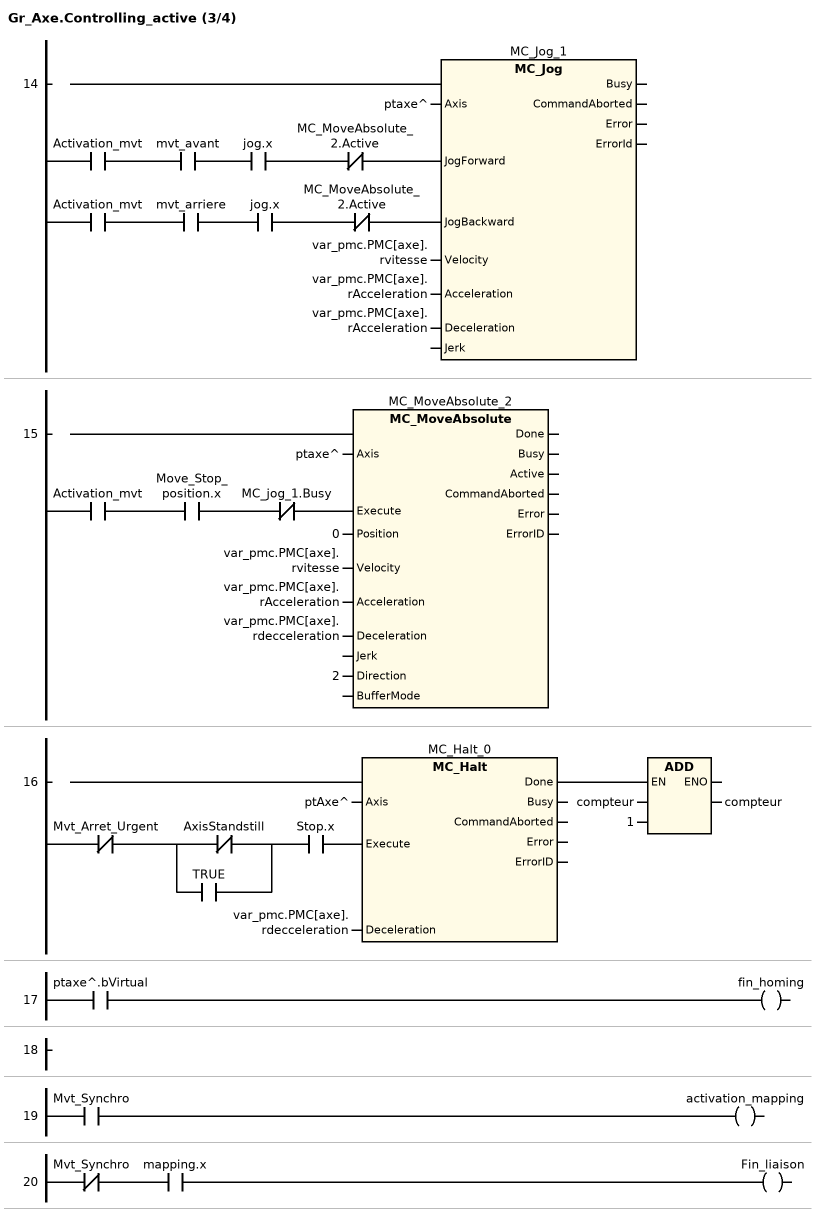
// NETWORK 14
MC_Jog_1(
    Axis := ptaxe^,
    JogForward := Activation_mvt AND mvt_avant AND jog.x AND NOT MC_MoveAbsolute_2.Active,
    JogBackward := Activation_mvt AND mvt_arriere AND jog.x AND NOT MC_MoveAbsolute_2.Active,
    Velocity := var_pmc.PMC[axe].rvitesse,
    Acceleration := var_pmc.PMC[axe].rAcceleration,
    Deceleration := var_pmc.PMC[axe].rAcceleration); // MC_Jog

// NETWORK 15
MC_MoveAbsolute_2(
    Axis := ptaxe^,
    Execute := Activation_mvt AND Move_Stop_position.x AND NOT MC_jog_1.Busy,
    Position := 0,
    Velocity := var_pmc.PMC[axe].rvitesse,
    Acceleration := var_pmc.PMC[axe].rAcceleration,
    Deceleration := var_pmc.PMC[axe].rdecceleration,
    Direction := 2); // MC_MoveAbsolute

// NETWORK 16
MC_Halt_0(
    Axis := ptAxe^,
    Execute := NOT Mvt_Arret_Urgent AND (NOT AxisStandstill OR TRUE) AND Stop.x,
    Deceleration := var_pmc.PMC[axe].rdecceleration); // MC_Halt
IF MC_Halt_0.Done THEN compteur := compteur + 1; END_IF

// NETWORK 17
fin_homing := ptaxe^.bVirtual;

// NETWORK 18

// NETWORK 19
activation_mapping := Mvt_Synchro;

// NETWORK 20
Fin_liaison := NOT Mvt_Synchro AND mapping.x;

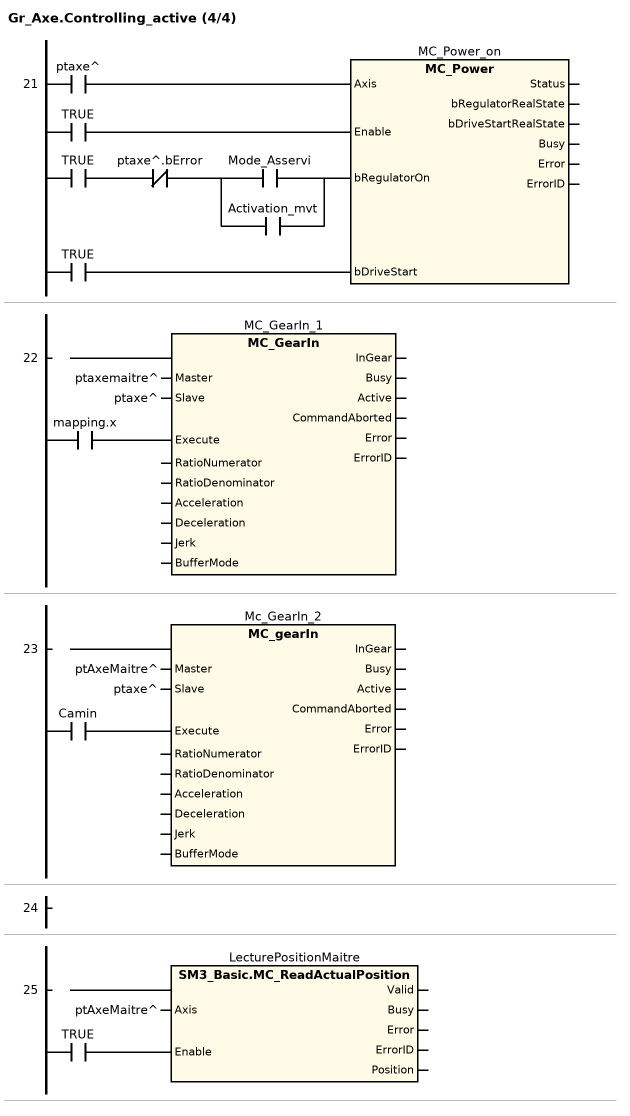
// NETWORK 21
MC_Power_on(
    Axis := ptaxe^,
    Enable := TRUE,
    bRegulatorOn := TRUE AND NOT ptaxe^.bError AND (Mode_Asservi OR Activation_mvt),
    bDriveStart := TRUE); // MC_Power

// NETWORK 22
MC_GearIn_1(Master := ptaxemaitre^, Slave := ptaxe^, Execute := mapping.x); // MC_GearIn

// NETWORK 23
Mc_GearIn_2(Master := ptAxeMaitre^, Slave := ptaxe^, Execute := Camin); // MC_gearIn

// NETWORK 24

// NETWORK 25
LecturePositionMaitre(Axis := ptAxeMaitre^, Enable := TRUE); // SM3_Basic.MC_ReadActualPosition
END_ACTION

ACTION Homing_active:
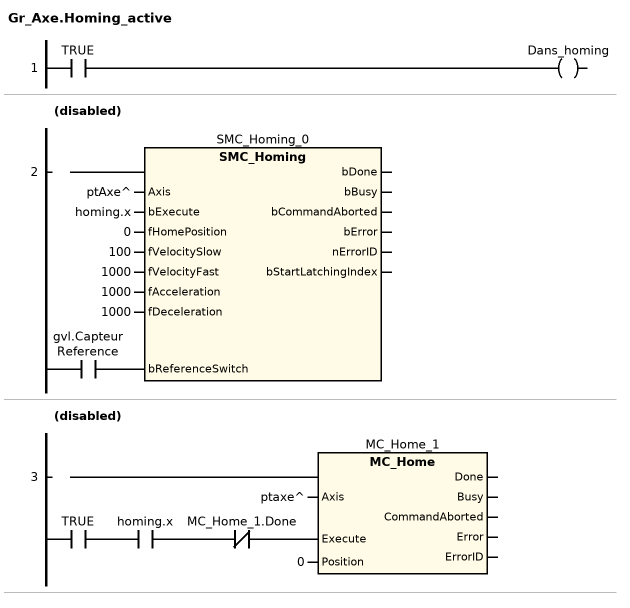
// NETWORK 1
Dans_homing := TRUE;

// NETWORK 2 (disabled)
// SMC_Homing_0(
//     Axis := ptAxe^,
//     bExecute := homing.x,
//     fHomePosition := 0,
//     fVelocitySlow := 100,
//     fVelocityFast := 1000,
//     fAcceleration := 1000,
//     fDeceleration := 1000,
//     bReferenceSwitch := gvl.CapteurReference); // SMC_Homing

// NETWORK 3 (disabled)
// MC_Home_1(Axis := ptaxe^, Execute := TRUE AND homing.x AND NOT MC_Home_1.Done, Position := 0); // MC_Home
END_ACTION

ACTION Jog_active:
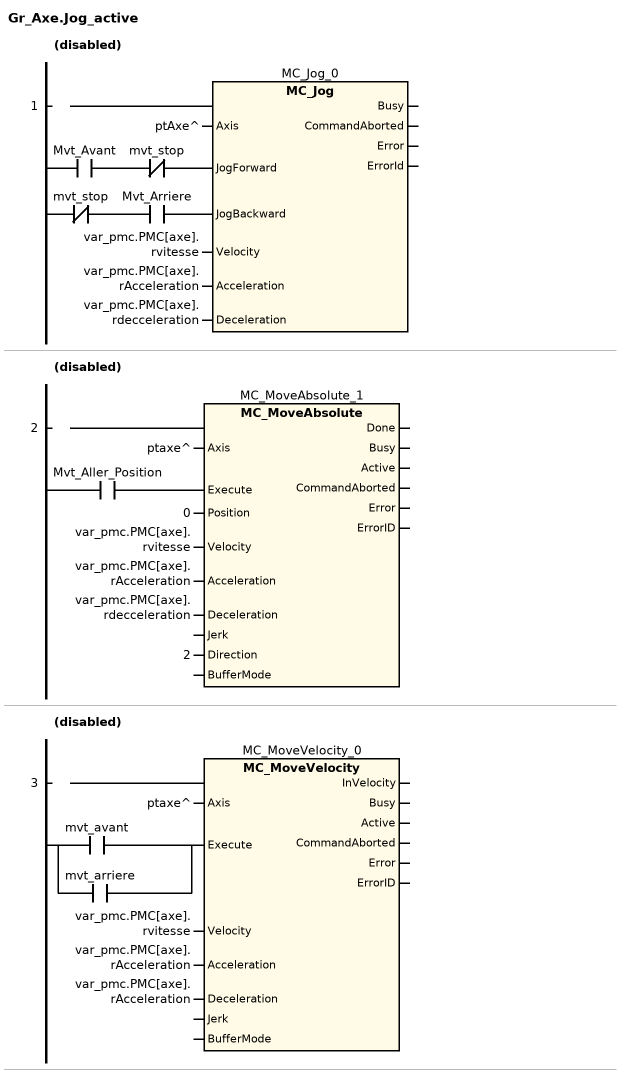
// NETWORK 1 (disabled)
// MC_Jog_0(
//     Axis := ptAxe^,
//     JogForward := Mvt_Avant AND NOT mvt_stop,
//     JogBackward := NOT mvt_stop AND Mvt_Arriere,
//     Velocity := var_pmc.PMC[axe].rvitesse,
//     Acceleration := var_pmc.PMC[axe].rAcceleration,
//     Deceleration := var_pmc.PMC[axe].rdecceleration); // MC_Jog

// NETWORK 2 (disabled)
// MC_MoveAbsolute_1(
//     Axis := ptaxe^,
//     Execute := Mvt_Aller_Position,
//     Position := 0,
//     Velocity := var_pmc.PMC[axe].rvitesse,
//     Acceleration := var_pmc.PMC[axe].rAcceleration,
//     Deceleration := var_pmc.PMC[axe].rdecceleration,
//     Direction := 2); // MC_MoveAbsolute

// NETWORK 3 (disabled)
// MC_MoveVelocity_0(
//     Axis := ptaxe^,
//     Execute := mvt_avant OR mvt_arriere,
//     Velocity := var_pmc.PMC[axe].rvitesse,
//     Acceleration := var_pmc.PMC[axe].rAcceleration,
//     Deceleration := var_pmc.PMC[axe].rAcceleration); // MC_MoveVelocity
END_ACTION

ACTION mapping_active:
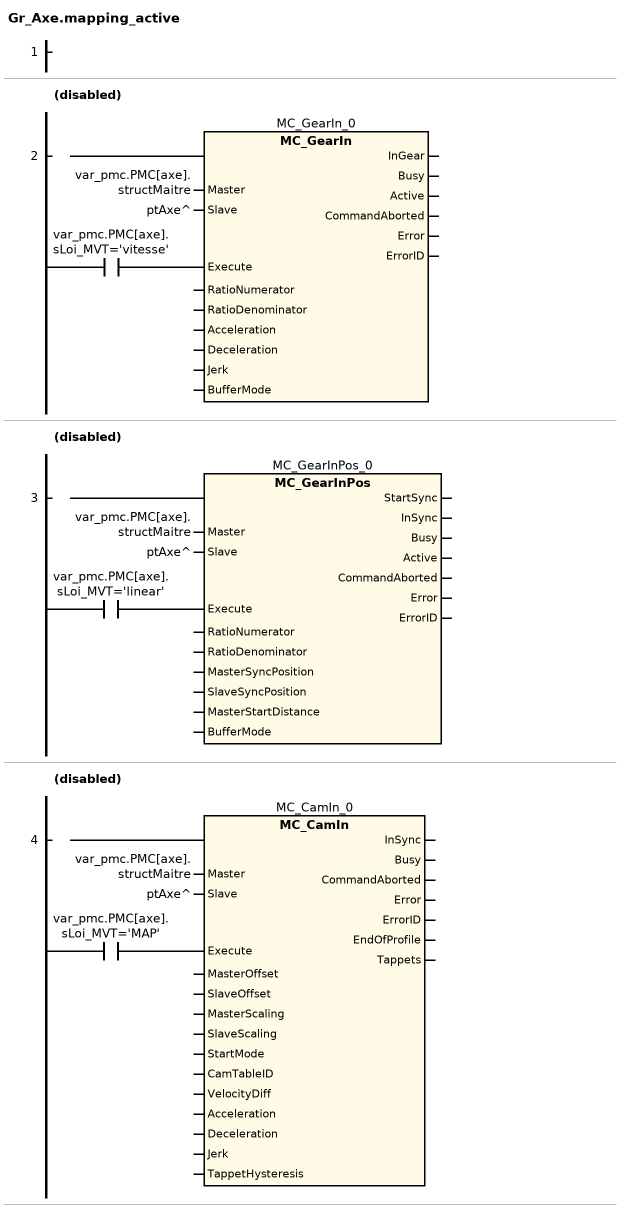
// NETWORK 1

// NETWORK 2 (disabled)
// MC_GearIn_0(
//     Master := var_pmc.PMC[axe].structMaitre,
//     Slave := ptAxe^,
//     Execute := var_pmc.PMC[axe].sLoi_MVT='vitesse'); // MC_GearIn

// NETWORK 3 (disabled)
// MC_GearInPos_0(
//     Master := var_pmc.PMC[axe].structMaitre,
//     Slave := ptAxe^,
//     Execute := var_pmc.PMC[axe].sLoi_MVT='linear'); // MC_GearInPos

// NETWORK 4 (disabled)
// MC_CamIn_0(
//     Master := var_pmc.PMC[axe].structMaitre,
//     Slave := ptAxe^,
//     Execute := var_pmc.PMC[axe].sLoi_MVT='MAP'); // MC_CamIn
END_ACTION

ACTION Move_Stop_position_active:
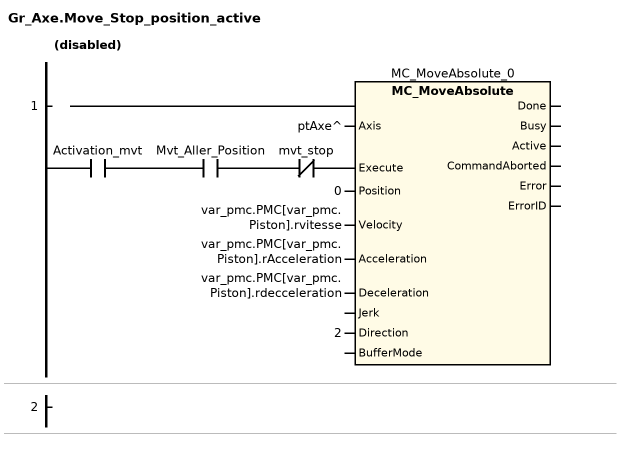
// NETWORK 1 (disabled)
// MC_MoveAbsolute_0(
//     Axis := ptAxe^,
//     Execute := Activation_mvt AND Mvt_Aller_Position AND NOT mvt_stop,
//     Position := 0,
//     Velocity := var_pmc.PMC[var_pmc.Piston].rvitesse,
//     Acceleration := var_pmc.PMC[var_pmc.Piston].rAcceleration,
//     Deceleration := var_pmc.PMC[var_pmc.Piston].rdecceleration,
//     Direction := 2); // MC_MoveAbsolute

// NETWORK 2
END_ACTION

ACTION Polling_active:
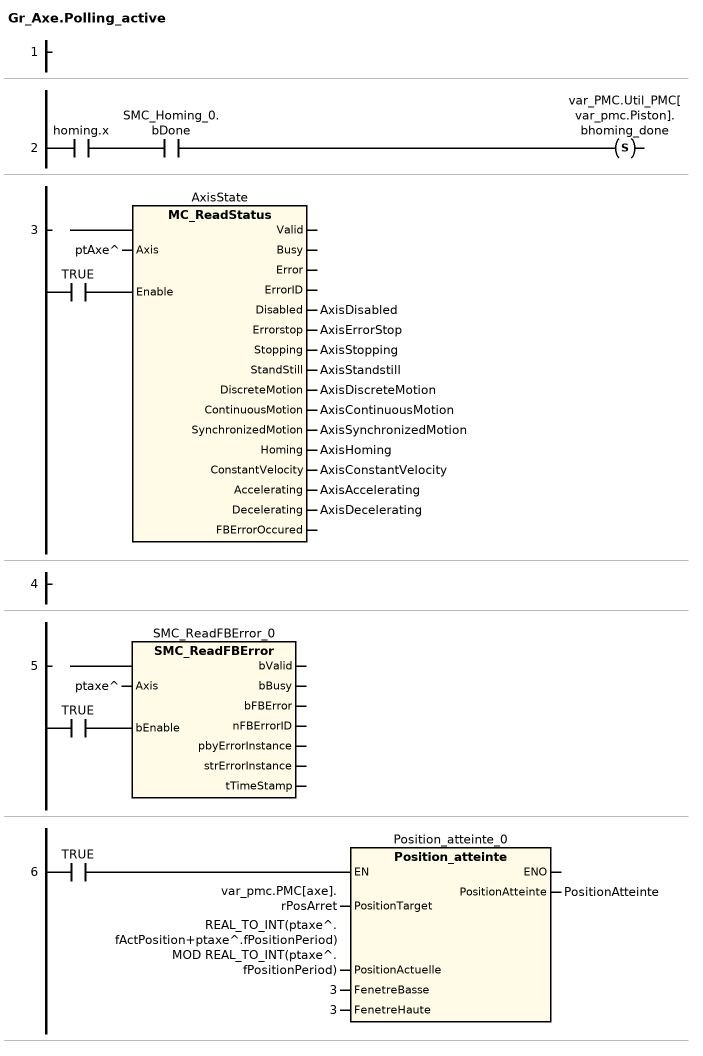
// NETWORK 1

// NETWORK 2
var_PMC.Util_PMC[var_pmc.Piston].bhoming_done S= homing.x AND SMC_Homing_0.bDone;

// NETWORK 3
AxisState(
    Axis := ptAxe^,
    Enable := TRUE,
    Disabled => AxisDisabled,
    Errorstop => AxisErrorStop,
    Stopping => AxisStopping,
    StandStill => AxisStandstill,
    DiscreteMotion => AxisDiscreteMotion,
    ContinuousMotion => AxisContinuousMotion,
    SynchronizedMotion => AxisSynchronizedMotion,
    Homing => AxisHoming,
    ConstantVelocity => AxisConstantVelocity,
    Accelerating => AxisAccelerating,
    Decelerating => AxisDecelerating); // MC_ReadStatus

// NETWORK 4

// NETWORK 5
SMC_ReadFBError_0(Axis := ptaxe^, bEnable := TRUE); // SMC_ReadFBError

// NETWORK 6
Position_atteinte_0(
    PositionTarget := var_pmc.PMC[axe].rPosArret,
    PositionActuelle := REAL_TO_INT(ptaxe^.fActPosition+ptaxe^.fPositionPeriod) MOD REAL_TO_INT(ptaxe^.fPositionPeriod),
    FenetreBasse := 3,
    FenetreHaute := 3,
    PositionAtteinte => PositionAtteinte); // Position_atteinte
END_ACTION

ACTION SetChannelParameters_active:
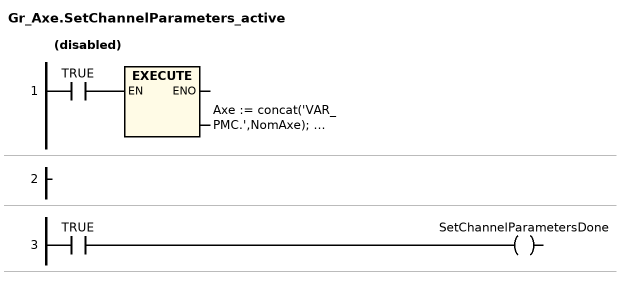
// NETWORK 1 (disabled)
// Axe := concat('VAR_PMC.',NomAxe);

// NETWORK 2

// NETWORK 3
SetChannelParametersDone := TRUE;
END_ACTION

ACTION Stop_active:
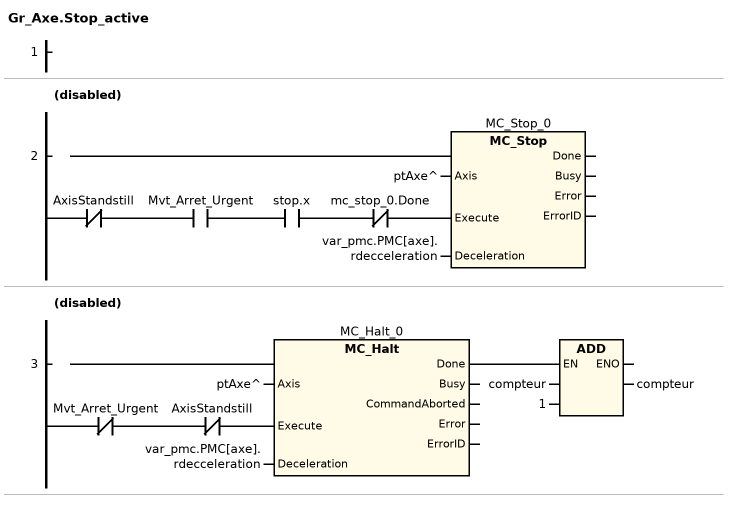
// NETWORK 1

// NETWORK 2 (disabled)
// MC_Stop_0(
//     Axis := ptAxe^,
//     Execute := NOT AxisStandstill AND Mvt_Arret_Urgent AND stop.x AND NOT mc_stop_0.Done,
//     Deceleration := var_pmc.PMC[axe].rdecceleration); // MC_Stop

// NETWORK 3 (disabled)
// MC_Halt_0(
//     Axis := ptAxe^,
//     Execute := NOT Mvt_Arret_Urgent AND NOT AxisStandstill,
//     Deceleration := var_pmc.PMC[axe].rdecceleration); // MC_Halt
// IF MC_Halt_0.Done THEN compteur := compteur + 1; END_IF
END_ACTION

END_FUNCTION_BLOCK

// Utilitaires/Position_atteinte
FUNCTION_BLOCK Position_atteinte
VAR_INPUT
	PositionTarget:REAL;
	PositionActuelle:REAL;
	FenetreBasse:REAL;
	FenetreHaute:REAL;
END_VAR
VAR_OUTPUT
	PositionAtteinte:BOOL;
END_VAR
VAR
END_VAR

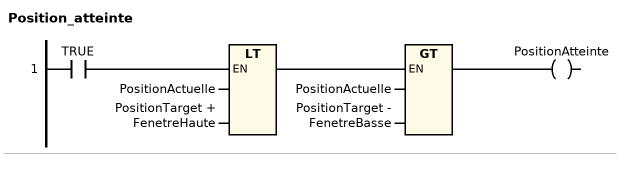
// NETWORK 1
PositionAtteinte := PositionActuelle < (PositionTarget + FenetreHaute) AND PositionActuelle > (PositionTarget - FenetreBasse);

END_FUNCTION_BLOCK

// Tests/ChoixOpMode
PROGRAM ChoixOpMode
VAR
	
END_VAR
VAR_INPUT
	ChoixMode:SINT;
END_VAR
VAR_OUTPUT
	OpModeActuel:sint;	
END_VAR


IF choixMode <> GVL.OpModeStober THEN
	GVL.OpModeStober := ChoixMode;
	OpModeActuel:=GVL.OpModeStober;
	ELSE
		RETURN;
END_IF

END_PROGRAM

// Accessoires/type_axe
FUNCTION_BLOCK type_axe
(* permet de définir si l'axe  est un :
														 CODEUR
														 VIRTUEL
														 MOTEUR   géré avec PSSU et retour codeur CAN sur PSSU
														 MOTEUR   géré avec PSSU et retour codeur sur PMCprimoMC ouC2
														 MOTEUR   géré avec drive au travers d'un réseau CAN ou ETHERCAT *)
VAR_INPUT

	udinumero: UDINT;
	udiindex:udint;
	
	END_VAR
VAR_OUTPUT

	bVirtuel: BOOL;
	bCodeur: BOOL;
	bDrive_PSSU_et_codeur_CAN: BOOL;
	bDrive_PSSU_et_codeur_PMCprimoC: BOOL;
	bDrive_CAN_Ethercat: BOOL;
	smoteur_utilise:STRING;
	Boucle_codeur_externe:bool;
END_VAR
VAR
type_drive_present: Type_drive_present;
	
	quels_moteurs: quels_moteurs;

	berreur1_config_axe:BOOL;
	berreur2_config_axe:BOOL;
	berreur3_config_axe:BOOL;
	berreur4_config_axe:BOOL;
	berreur5_config_axe:BOOL;
	
	bVirtuel1:BOOL;
	bVirtuel2:BOOL;
	bVirtuel3:BOOL;
	bVirtuel4:BOOL;
	bVirtuel5:BOOL;

END_VAR


		(*=== tests si SMoteur est un Virtuel , un codeur  ===*)
		
		type_drive_present(		udinumero:= udinumero,udiindex:=udiindex); 
		
		var_infor.info[udinumero,udiindex].berror:=0;
		var_infor.info[udinumero,udiindex].smoteur_utilise:=var_PMC.PMC[udinumero,udiindex].SMoteur;
	
		(* === bcodeur ===*)
		Boucle_codeur_externe:=var_pmc.Spec_PMC[udinumero,udiindex].Boucle_codeur_externe ;
		bCodeur    :=var_PMC.PMC[udinumero,udiindex].SMoteur      =          'CODEUR' AND NOT(type_drive_present.presence_drive)  ;
		berreur1_config_axe:= var_PMC.PMC[udinumero,udiindex].SMoteur      =          'CODEUR' AND (type_drive_present.presence_drive=TRUE)  ;
		smoteur_utilise:=var_PMC.PMC[udinumero,udiindex].SMoteur;
		
		bVirtuel1      :=berreur1_config_axe;
		
		
			var_infor.info[udinumero,udiindex].bCodeur:=(bCodeur =TRUE);
		
		
			(* === bvirtuel ===*)
			bVirtuel2      :=var_PMC.PMC[udinumero,udiindex].SMoteur      =          'VIRTUEL';
		
			bVirtuel3:=( type_drive_present.presence_drive=FALSE)AND (bCodeur=FALSE)   OR ( type_drive_present.presence_drive=TRUE) AND (bCodeur =TRUE);
			berreur2_config_axe:=( type_drive_present.presence_drive=FALSE)AND (bCodeur=FALSE)   OR ( type_drive_present.presence_drive=TRUE) AND (bCodeur =TRUE);
		
			bVirtuel4:= ( type_drive_present.presence_drive=FALSE)AND var_PMC.PMC[udinumero,udiindex].SMoteur <> 'CODEUR' AND var_PMC.PMC[udinumero,udiindex].SMoteur <> 'VIRTUEL';
			berreur3_config_axe:=( type_drive_present.presence_drive=FALSE)AND var_PMC.PMC[udinumero,udiindex].SMoteur <> 'CODEUR' AND var_PMC.PMC[udinumero,udiindex].SMoteur <> 'VIRTUEL';
		
			quels_moteurs (smoteur:=var_PMC.PMC[udinumero,udiindex].SMoteur );
			bVirtuel5:=quels_moteurs.virtuel;

			bVirtuel:= bVirtuel1 OR bVirtuel2 OR bVirtuel3 OR bVirtuel4 OR bVirtuel5;
			
			var_infor.info[udinumero,udiindex].bVirtuel:=(bVirtuel=TRUE);
			
			IF (bVirtuel =TRUE) THEN var_infor.info[udinumero,udiindex].smoteur_utilise:='VIRTUEL'; END_IF;
	
	
			(* ===  drive ProtegoD, PMCtendoDD5 ou au travers de PSSU ===*)
			(* === avec codeur CAN  9<= FS <=10  et  sMoteur ='MOTEUR' ===*)
			bDrive_PSSU_et_codeur_CAN:= ( (var_PMC.PMC[udinumero,udiindex].Mode_Asservissement>=9 AND var_PMC.PMC[udinumero,udiindex].Mode_Asservissement<=10) AND NOT(bCodeur) AND NOT(bVirtuel));
			var_infor.info[udinumero,udiindex].bDrive_PSSU_et_codeur_CAN:= (bDrive_PSSU_et_codeur_CAN=TRUE);
		
			(* === avec codeur incrémental ou SSI   0<= FS <=8   et  sMoteur ='MOTEUR' ===*)
			//bDrive_PSSU_et_codeur_PMCprimoC:= ( (var_PMC.PMC[udinumero,udiindex].Mode_Asservissement>=0 AND var_PMC.PMC[udinumero,udiindex].Mode_Asservissement<=8) AND NOT(bCodeur) AND NOT(bVirtuel));
			//var_infor.info[udinumero,udiindex].bDrive_PSSU_et_codeur_PMCprimoC:=(bDrive_PSSU_et_codeur_PMCprimoC=TRUE);
		
			(*=== avec drive reconnu sur réseau CAN et/ou Ethercat    19<= FS <=35 *)
			bDrive_CAN_Ethercat:=(var_PMC.PMC[udinumero,udiindex].Mode_Asservissement>=19 AND var_PMC.PMC[udinumero,udiindex].Mode_Asservissement<=35) AND NOT(bVirtuel) AND NOT(bCodeur) AND (type_drive_present.presence_drive=TRUE);
			var_infor.info[udinumero,udiindex].bDrive_CAN_Ethercat:=(bDrive_CAN_Ethercat=TRUE);
		
			
			var_infor.info[udinumero,udiindex].bError:= berreur1_config_axe OR berreur2_config_axe OR berreur3_config_axe;
			
			IF(var_infor.info[udinumero,udiindex].bError=TRUE) THEN		var_infor.info[udinumero,udiindex].iErrorNumber:=507; END_IF;

END_FUNCTION_BLOCK

// EtherCAT/EsclavesReady
//Détermine si les esclaves EtherCAT inscrits dans la liste des appareils sont prêts à fonctionner

FUNCTION_BLOCK EsclavesReady
VAR_INPUT
END_VAR
VAR_OUTPUT
END_VAR
VAR
	ListeEtats:ARRAY [0..gvl_ethercat.EtherCATSlavesNumber] OF BUS_STATE;
	index : INT :=0;
END_VAR

FOR index :=0 TO GVL_EtherCAT.EtherCATSlavesNumber BY 1 DO
	ListeEtats[index]:=GVL_EtherCAT.ListeEtherCATSlaves[index].wState;
END_FOR

END_FUNCTION_BLOCK

// /Visualization
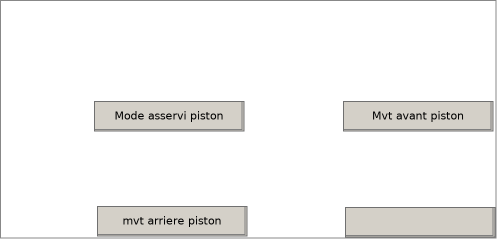
VISUALIZATION Visualization  // 497x239
    Button (94,101 150x30), "Mode asservi piston"
        toggle Gestion_axes.Gr_Piston.Mode_Asservi
    Button (343,101 150x30), "Mvt avant piston"
        toggle Gestion_axes.Gr_Piston.Mvt_Avant
    Button (97,206 150x30), "mvt arriere piston"
        toggle Gestion_axes.Gr_Piston.Mvt_Arriere
    Button (345,207 150x30)
END_VISUALIZATION

// /VisualizationAxe1
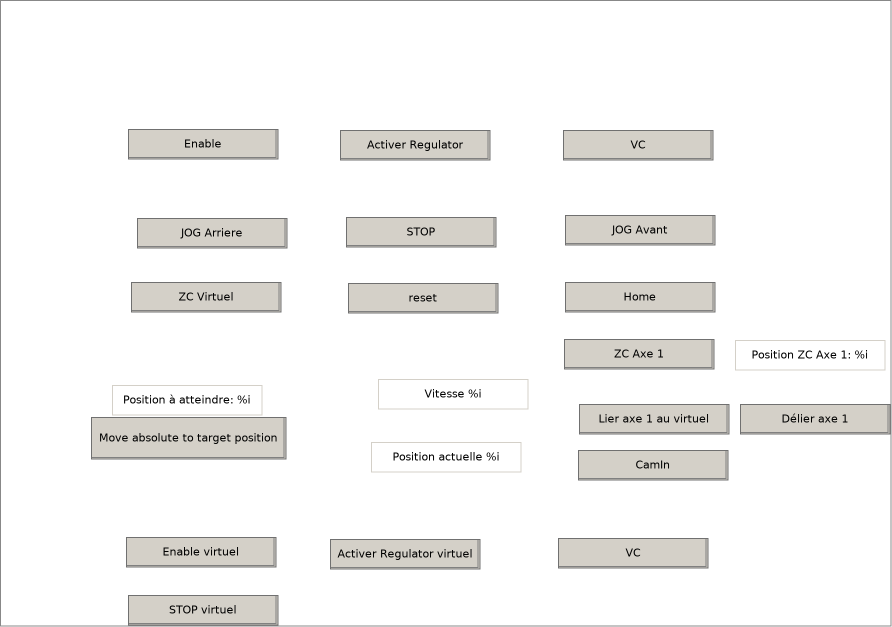
VISUALIZATION VisualizationAxe1  // 892x627
    Button (128,129 150x30), "Enable"
        toggle plc_prg.EnableAxe1
    Button (340,130 150x30), "Activer Regulator"
        toggle PLC_PRG.ActiverRegulateurAxe1
    Button (563,130 150x30), "VC"
        toggle plc_prg.VC_axe1
    Button (348,283 150x30), "reset"
        toggle plc_prg.ResetAxe1
    Button (346,217 150x30), "STOP"
        toggle plc_prg.StopAxe1
    Button (565,215 150x30), "JOG Avant"
        toggle plc_prg.JOGAvant
    Button (137,218 150x30), "JOG Arriere"
        toggle plc_prg.JOGArriere
    Textfield (112,385 150x30), "Position à atteindre: %i", text variable: GVL.TargetAbsolutePosition
        OnMouseClick: write the text variable via Default, min 0, max 50000
    Button (91,417 195x42), "Move absolute to target position"
        toggle plc_prg.MoveAbsolute
    Textfield (378,379 150x30), "Vitesse %i", text variable: GVL.Speed
        OnMouseClick: write GVL.Speed via Default, min 0, max 500000
    Button (565,282 150x30), "Home"
        toggle plc_prg.Home
    Button (131,282 150x30), "ZC Virtuel"
        toggle plc_prg.ZC_Virtuel
    Button (564,339 150x30), "ZC Axe 1"
        toggle plc_prg.ZC_Axe1
    Textfield (735,340 150x30), "Position ZC Axe 1: %i", text variable: GVL.Position_ZC_Axe_1
        OnMouseClick: write GVL.Position_ZC_Axe_1 via Default, min -50000, max 50000
    Button (579,404 150x30), "Lier axe 1 au virtuel"
        toggle plc_prg.XM
    Button (578,450 150x30), "CamIn"
        toggle plc_prg.CamIn
    Button (740,404 150x30), "Délier axe 1"
        toggle plc_prg.GearOut
    Textfield (371,442 150x30), "Position actuelle %i", text variable: PLC_prg.MC_ReadActualPosition_0.Position
    Button (126,537 150x30), "Enable virtuel"
        toggle PLC_PRG.enable_virtuel
    Button (330,539 150x30), "Activer Regulator virtuel"
        toggle plc_prg.activer_regulator
    Button (558,538 150x30), "VC"
        toggle plc_prg.VC_virtuel
    Button (128,595 150x30), "STOP virtuel"
        toggle plc_prg.MCSTOP
END_VISUALIZATION

// /VisualizationCamIn
VISUALIZATION VisualizationCamIn  // 2x2
END_VISUALIZATION

// /VisualizationVirtuel
